(* Schneider Machine Expert - Basic project Slave 1 AHU Mod  TCP, file version 2.2.0.0 *)
(* ProjectInformations: Name=New project *)

HARDWARE
  Cpu 0: TM221ME16R/G
  ModuleExtensionObject 0: TM3DI16/G
  ModuleExtensionObject 1: TM3DQ16R/G
  ModuleExtensionObject 2: TM3AI8/G
  ModuleExtensionObject 3: TM3AQ4/G
  ModuleExtensionObject 4: TM3AQ2/G
  EthernetConfiguration: NetworkName=M221, IpAllocationMode=FixedAddress, IpAddress=10.3.12.251, SubnetMask=255.255.252.0
  SerialLineConfiguration: Baud=Baud9600, Parity=ParityEven, DataBits=DataBits8, StopBits=StopBits1, PhysicalMedium=PhysicalMediumRs485, TransmissionMode=TransmissionModeModbusRtu, SlaveId=1, Addressing=MasterAddressing
  MastTask: UsePeriodScanMode=false, PeriodScan=100
  FastTask: Period=255
  CpuBehavior: StartingMode=StartAsPreviousState, AutoSaveRamOnEeprom=true, WatchdogPeriod=250

SYMBOLS  (address, symbol, comment, settings)
  %M0       STRINV1  "Start Inverter AHU Line 09-10"
  %M1       STPINV1  "Stop Inverter AHU Line 09-10"
  %M2       OPNDMPR1  "Open Damper AHU Line 09-10"
  %M3       CLODMPR1  "Close Damper AHU Line 09-10"
  %M4       S_REMOTE_1  "Selector REMOTE MODE !!! Line 09-10"
  %M5       S_LOCAL_1  "Selector LOCAL MODE !!! Line 09-10"
  %M6       STRINV2  "Start Inverter AHU Line 11-12"
  %M7       STPINV2  "Stop Inverter AHU Line 11-12"
  %M8       OPNDMPR2  "Open Damper AHU Line 11-12"
  %M9       CLODMPR2  "Close Damper AHU Line 11-12"
  %M10      S_REMOTE_2  "Selector REMOTE MODE !!! Line 11-12"
  %M11      STRINV3  "Start Inverter AHU Line 17-18"
  %M12      STPINV3  "Stop Inverter AHU Line 17-18"
  %M13      OPNDMPR3  "Open Damper AHU Line 17-18"
  %M14      CLODMPR3  "Close Damper AHU Line 17-18"
  %M15      S_REMOTE_3  "Selector REMOTE MODE !!! Line 17-18"
  %M16      INPUT_ONINV_1  "On Inverter AHU Line 09-10"
  %M17      INPUT_ONINV_2  "On Inverter AHU Line 11-12"
  %M18      INPUT_ONINV_3  "On Inverter AHU Line 17-18"
  %M19      INPUT_ALARM_1  "Alarm Inverter AHU Line 09-10"
  %M20      INPUT_ALARM_2  "Alarm Inverter AHU Line 11-12"
  %M21      INPUT_ALARM_3  "Alarm Inverter AHU Line 17-18"
  %M22      S_LOCAL_2  "Selector LOCAL MODE !!! Line 11-12"
  %M23      S_LOCAL_3  "Selector LOCAL MODE !!! Line 17-18"
  %M31      ALARM1  "ALARM AHU LINE 09-10 ON !!!!"
  %M32      ALARM2  "ALARM AHU LINE 11-12 ON !!!!"
  %M33      ALARM3  "ALARM AHU LINE 17-18 ON !!!!"
  %M34      RUN_1  "RUN AHU LINE 09-10"
  %M35      RUN_2  "RUN AHU LINE 11-12"
  %M36      RUN_3  "RUN AHU LINE 17-18"
  %M37      INV_1_ON  "INVERTER AHU LINE 09-10 ON !!!"
  %M38      INV_2_ON  "INVERTER AHU LINE 11-12 ON !!!"
  %M39      INV_3_ON  "INVERTER AHU LINE 17-18 ON !!!"
  %M61      FLAG_MAN_INV1  "INVERTER LINE 09-10 ON !!! MANUAL"
  %M62      FLAG_MAN_DMPR1  "DAMPER LINE 09-10 ON !!! MANUAL"
  %M63      FLAG_AUTO_INV1  "INVERTER LINE 09-10 ON !!! AUTO"
  %M64      FLAG_MAN_INV2  "INVERTER LINE 11-12 ON !!! MANUAL"
  %M65      FLAG_MAN_DMPR2  "DAMPER LINE 11-12 ON !!! MANUAL"
  %M66      FLAG_AUTO_INV2  "INVERTER LINE 11-12 ON !!! AUTO"
  %M67      FLAG_MAN_INV3  "INVERTER LINE 17-18 ON !!! MANUAL"
  %M68      FLAG_MAN_DMPR3  "DAMPER LINE 17-18 ON !!! MANUAL"
  %M69      FLAG_AUTO_INV3  "INVERTER LINE 17-18 ON !!! AUTO"
  %M82      FLAG_AUTO_DMPR_1  "DAMPER LINE 09-10 ON !!! AUTO"
  %M83      FLAG_AUTO_DMPR_2  "DAMPER LINE 11-12 ON !!! AUTO"
  %M84      FLAG_AUTO_DMPR_3  "DAMPER LINE 17-18 ON !!! AUTO"
  %M85      ALARM_MODBUS  "MODBUS COMMUNICATION ERROR !!! CHECK CONNECTION"
  %M86      REMOTE_START_INV_1  "REMOTE Start Inverter AHU Line 09-10"
  %M87      REMOTE_STOP_INV_1  "REMOTE Stop Inverter AHU Line 09-10"
  %M88      REMOTE_START_DMPR_1  "REMOTE Open Damper AHU Line 09-10"
  %M89      REMOTE_STOP_DMPR_1  "REMOTE Close Damper AHU Line 09-10"
  %M90      REMOTE_START_INV_2  "REMOTE Start Inverter AHU Line 11-12"
  %M91      REMOTE_STOP_INV_2  "REMOTE Stop Inverter AHU Line 11-12"
  %M92      REMOTE_START_DMPR_2  "REMOTE Open Damper AHU Line 11-12"
  %M93      REMOTE_STOP_DMPR_2  "REMOTE Close Damper AHU Line 11-12"
  %M94      REMOTE_START_INV_3  "REMOTE Start Inverter AHU Line 17-18"
  %M95      REMOTE_STOP_INV_3  "REMOTE Stop Inverter AHU Line 17-18"
  %M96      REMOTE_START_DMPR_3  "REMOTE Open Damper AHU Line 17-18"
  %M97      REMOTE_STOP_DMPR_3  "REMOTE Close Damper AHU Line 17-18"
  %M100     MANUAL_AUTO_1  "REMOTE OPTION MODE AHU LINE 09-10"
  %M101     MANUAL_AUTO_2  "REMOTE OPTION MODE AHU LINE 11-12"
  %M102     MANUAL_AUTO_3  "REMOTE OPTION MODE AHU LINE 17-18"
  %M103     DMPR_1_ON  "DAMPER LINE 09-10 ON !!!"
  %M104     DMPR_2_ON  "DAMPER LINE 11-12 ON !!!"
  %M105     DMPR_3_ON  "DAMPER LINE 17-18 ON !!!"
  %M106     ERR_SERIAL_1  "Serial Comunication Error 1"
  %M107     ERR_SERIAL_2  "Serial Communication Error 2"
  %M119     RESET_ALARM
  %M120     TEMP_1_HIGH
  %M121     TEMP_1_LOW
  %M122     HUM_1_HIGH
  %M123     HUM_1_LOW
  %M124     PRESS_1_HIGH
  %M125     PRESS_1_LOW
  %M130     TEMP_2_HIGH
  %M131     TEMP_2_LOW
  %M132     HUM_2_HIGH
  %M133     HUM_2_LOW
  %M134     PRESS_2_HIGH
  %M135     PRESS_2_LOW
  %M140     TEMP_3_HIGH
  %M141     TEMP_3_LOW
  %M142     HUM_3_HIGH
  %M143     HUM_3_LOW
  %M144     PRESS_3_HIGH
  %M145     PRESS_3_LOW
  %S6       SB_TB1S  "Time base of 1 s generated by an internal clock"
  %S12      SB_RUNMODE  "The controller is running"
  %MW9      AI_SCALE_DIFF_PRESSURE_1  "Memory Hasil Scalling Analog Input Differensial Pressure Line 09-10"
  %MW11     AO1_LO_LIMIT
  %MW12     AO1_HI_LIMIT
  %MW13     AO2_LO_LIMIT
  %MW14     AO2_HI_LIMIT
  %MW15     AO3_LO_LIMIT
  %MW16     AO3_HI_LIMIT
  %MW30     AI_SCALE_DIFF_PRESSURE_2
  %MW51     AI_SCALE_DIFF_PRESSURE_3
  %MW73     AI_SCALE_TEMP_1
  %MW95     AI_SCALE_HUMIDITY_1
  %MW117    AO_SCALE_TEMP_1
  %MW139    AO_SCALE_TEMP_2
  %MW161    AO_SCALE_TEMP_3
  %MW183    AO_SCALE_HUMIDITY_1
  %MW205    AO_SCALE_HUMIDITY_2
  %MW227    AO_SCALE_HUMIDITY_3
  %MW251    TEMP_1_SETPOINT
  %MW252    TEMP_1_P
  %MW253    TEMP_1_I
  %MW254    TEMP_1_D
  %MW255    TEMP_1_SAMPLING
  %MW256    SET_SPEED_INV_1
  %MW257    ALRM_TEMP1_LOW_SET
  %MW258    ALRM_TEMP1_HIGH_SET
  %MW259    ALRM_PRESS1_LOW_SET
  %MW260    ALRM_PRESS1_HIGH_SET
  %MW281    TEMP_2_SETPOINT
  %MW282    TEMP_2_P
  %MW283    TEMP_2_I
  %MW284    TEMP_2_D
  %MW285    TEMP_2_SAMPLING
  %MW286    SET_SPEED_INV_2
  %MW287    ALRM_TEMP_2_LOW_SET
  %MW288    ALRM_TEMP_2_HIGH_SET
  %MW289    ALRM_PRESS2_LOW_SET
  %MW290    ALRM_PRESS2_HIGH_SET
  %MW311    TEMP_3_SETPOINT
  %MW312    TEMP_3_P
  %MW313    TEMP_3_I
  %MW314    TEMP_3_D
  %MW315    TEMP_3_SAMPLING
  %MW316    SET_SPEED_INV_3
  %MW317    ALRM_TEMP_3_LOW_SET
  %MW318    ALRM_TEMP_3_HIGH_SET
  %MW319    ALRM_PRESS3_LOW_SET
  %MW320    ALRM_PRESS3_HIGH_SET
  %MW341    HUMIDITY_1_SETPOINT
  %MW342    HUMIDITY_1_P
  %MW343    HUMIDITY_1_I
  %MW344    HUMIDITY_1_D
  %MW345    HUMIDITY_1_SAMPLING
  %MW346    SET_DAMPER_POSITION_1
  %MW347    ALRM_HUMIDITY_1_LOW_SET
  %MW348    ALRM_HUMIDITY_1_HIGH_SET
  %MW380    DMPR_1_VIEW
  %MW381    DMPR_2_VIEW
  %MW382    DMPR_3_VIEW
  %MW401    HUMIDITY_2_SETPOINT
  %MW402    HUMIDITY_2_P
  %MW403    HUMIDITY_2_I
  %MW404    HUMIDITY_2_D
  %MW405    HUMIDITY_2_SAMPLING
  %MW406    SET_DAMPER_2_POSITION
  %MW407    ALRM_HUMIDITY_2_LOW_SET
  %MW408    ALRM_HUMIDITY_2_HIGH_SET
  %MW431    HUMIDITY_3_SETPOINT
  %MW432    HUMIDITY_3_P
  %MW433    HUMIDITY_3_I
  %MW434    HUMIDITY_3_D
  %MW435    HUMIDITY_3_SAMPLING
  %MW436    SET_DAMPER_3_POSITION
  %MW437    ALRM_HUMIDITY_3_LOW_SET
  %MW438    ALRM_HUMIDITY_3_HIGH_SET
  %MW461    TEMP_1_DATA_SERIAL  "Data Temperature Line 09-10"
  %MW462    TEMP_2_DATA_SERIAL  "Data Temperature Line 11-12"
  %MW463    HUMIDITY_1_DATA_SERIAL  "Data Humidity Line 09-10"
  %MW464    HUMIDITY_2_DATA_SERIAL  "Data Humidity Line 11-12"
  %MW465    ERROR_DATA  "Error Communication"
  %MW480    AI_SCALE_TEMP_2
  %MW490    AI_SCALE_TEMP_3
  %MW500    AI_SCALE_HUMIDITY_2
  %MW510    AI_SCALE_HUMIDITY_3
  %MW520    AI_SCALE_DAMPER__POSITION_1
  %MW530    AI_SCALE_DAMPER_POSITION_2
  %MW540    AI_SCALE_DAMPER_POSITION_3
  %MW542    ALARM_WORD
  %MW600    HUMIDITY_LINE_1718  "Data serial humidity line 17-18"
  %MW601    TEMPERATURE_LINE_1718  "Data serial temperature line 17-18"
  %MW630    INV_1_HZ
  %MW640    INV_2_HZ
  %MW650    INV_3_HZ
  %READ_VAR0   [Link(Value(FBComLinkParameterEnums=SerialLine1)), RemoteDeviceId(Value(int=2)), Timeout(Value(int=100)), ObjType(Value(FBComObjTypeParameterEnums=IW)), FirstObj(Value(int=0)), Quantity(Value(int=1)), IndexData(Value(int=600))]
  %READ_VAR1   [Link(Value(FBComLinkParameterEnums=SerialLine1)), RemoteDeviceId(Value(int=3)), Timeout(Value(int=100)), ObjType(Value(FBComObjTypeParameterEnums=IW)), FirstObj(Value(int=0)), Quantity(Value(int=1)), IndexData(Value(int=601))]
  %RTC0     REAL_TIME_0  [Day(Value(int=1)), Month(Value(int=1)), Year(Value(int=2000)), Hours(Value(int=0)), Minutes(Value(int=0)), Seconds(Value(int=0))]
  %WRITE_READ_VAR0   [Link(Value(FBComLinkParameterEnums=EthernetLink)), RemoteDeviceId(Value(int=1)), Timeout(Value(int=100)), ObjType(Value(FBComObjTypeParameterEnums=MW)), FirstWriteObj(Value(int=10)), WriteQuantity(Value(int=1)), IndexDataOut(Value(int=465)), FirstReadObj(Value(int=0)), ReadQuantity(Value(int=4)), IndexDataIn(Value(int=461))]
  %I0.0     INV1_START  "LOCAL !!! Untuk mengontrol START Inverter AHU Line 09-10"
  %I0.1     INV1_STOP  "LOCAL !!! Untuk mengontrol STOP Inverter AHU Line 09-10"
  %I0.2     DMPR1_OPEN  "LOCAL !!! Untuk mengontrol OPEN Damper  AHU Line 09-10"
  %I0.3     DMPR1_CLOSE  "LOCAL !!! Untuk mengontrol CLOSE Damper  AHU Line 09-10"
  %I0.4     REMOTE_1  "SELECTOR SWITCH REMOTE !!! AHU LINE 09-10"
  %I0.5     LOCAL_1  "SELECTOR SWITCH LOCAL !!! AHU LINE 09-10"
  %I0.6     INV2_START  "LOCAL !!! Untuk mengontrol START Inverter AHU Line 11-12"
  %I0.7     INV2_STOP  "LOCAL !!! Untuk mengontrol STOP Inverter AHU Line 11-12"
  %Q0.0     ALARM_1  "Alarm Indikator Line 09-10"
  %Q0.1     ALARM_2  "Alarm Indikator Line 11-12"
  %Q0.2     ALARM_3  "Alarm Indikator Line 17-18"
  %Q0.3     RUN_STATUS_1  "Running Status Line 09-10"
  %Q0.4     RUN_STATUS_2  "Running Status Line 11-12"
  %Q0.5     RUN_STATUS_3  "Running Status Line 17-18"
  %Q0.6     INVERTER_1_ON  "Trigger Inverter Line 09-10"
  %Q0.7     INVERTER_2_ON  "Trigger Inverter Line 11-12"
  %I1.0     DMPR2_OPEN  "LOCAL !!! Untuk mengontrol OPEN Damper  AHU Line 11-12"
  %I1.1     DMPR2_CLOSE  "LOCAL !!! Untuk mengontrol CLOSE Damper  AHU Line 11-12"
  %I1.2     REMOTE_2  "SELECTOR SWITCH REMOTE !!! AHU LINE 11-12"
  %I1.3     INV3_START  "LOCAL !!! Untuk mengontrol START Inverter AHU Line 17-18"
  %I1.4     INV3_STOP  "LOCAL !!! Untuk mengontrol STOP Inverter AHU Line  17-18"
  %I1.5     DMPR3_OPEN  "LOCAL !!! Untuk mengontrol OPEN Damper  AHU Line 17-18"
  %I1.6     DMPR3_CLOSE  "LOCAL !!! Untuk mengontrol CLOSE Damper  AHU Line 17-18"
  %I1.7     REMOTE_3  "SELECTOR SWITCH REMOTE !!! AHU LINE 17-18"
  %I1.8     INPUTRUN1  "Signal Running Inverter AHU Line 09-10"
  %I1.9     INPUTRUN2  "Signal Running Inverter AHU Line 11-12"
  %I1.10    INPUTRUN3  "Signal Running Inverter AHU Line 17-18"
  %I1.11    ALARM1_INPUT  "Signal Alarm Inverter AHU Line 09-10"
  %I1.12    ALARM2_INPUT  "Signal Alarm Inverter AHU Line 11-12"
  %I1.13    ALARM3_INPUT  "Signal Alarm Inverter AHU Line 17-18"
  %I1.14    LOCAL_2  "SELECTOR SWITCH LOCAL !!! AHU LINE 11-12"
  %I1.15    LOCAL_3  "SELECTOR SWITCH LOCAL !!! AHU LINE 17-18"
  %Q2.0     INVERTER_3_ON  "Trigger Inverter Line 17-18"
  %IW3.0    PRESS_AHU_1  "Differensial Pressure Line 09-10"  [Type=Type_4_20mA, Scope=Scope_Customized, Minimum=4000, Maximum=20000]
  %IW3.1    PRESS_AHU_2  "Differensial Pressure Line 11-12"  [Type=Type_4_20mA, Scope=Scope_Customized, Minimum=4000, Maximum=20000]
  %IW3.2    PRESS_AHU_3  "Differensial Pressure Line 17-18"  [Type=Type_4_20mA, Scope=Scope_Customized, Minimum=4000, Maximum=20000]
  %IW3.3    SPARE1  [Type=Type_4_20mA, Scope=Scope_Customized, Minimum=4000, Maximum=20000]
  %IW3.4    SPARE2  [Type=Type_4_20mA, Scope=Scope_Customized, Minimum=4000, Maximum=20000]
  %IW3.5    DAMP_POS_AHU_1  "FeedBack Damper Position Line 09-10"  [Type=Type_0_10V, Scope=Scope_Customized, Minimum=0, Maximum=10000]
  %IW3.6    DAMP_POS_AHU_2  "FeedBack Damper Position Line 11-12"  [Type=Type_0_10V, Scope=Scope_Customized, Minimum=0, Maximum=10000]
  %IW3.7    DAMP_POS_AHU_3  "FeedBack Damper Position Line 17-18"  [Type=Type_0_10V, Scope=Scope_Customized, Minimum=0, Maximum=10000]
  %QW4.0    AO_INV_1  "Analog Output Speed Inverter Line 09-10"  [Type=Type_0_10V, Scope=Scope_Customized, Minimum=0, Maximum=10000]
  %QW4.1    AO_INV_2  "Analog Output Speed Inverter Line 11-12"  [Type=Type_0_10V, Scope=Scope_Customized, Minimum=0, Maximum=10000]
  %QW4.2    AO_INV_3  "Analog Output Speed Inverter Line 17-18"  [Type=Type_0_10V, Scope=Scope_Customized, Minimum=0, Maximum=10000]
  %QW4.3    AO_DMPR_1  "Analog Output Damper Control Line 09-10"  [Type=Type_0_10V, Scope=Scope_Customized, Minimum=0, Maximum=10000]
  %QW5.0    AO_DMPR_2  "Analog Output Damper Control Line 11-12"  [Type=Type_0_10V, Scope=Scope_Customized, Minimum=0, Maximum=10000]
  %QW5.1    AO_DMPR_3  "Analog Output Damper Control Line 17-18"  [Type=Type_0_10V, Scope=Scope_Customized, Minimum=0, Maximum=10000]

POU TRANSFER INPUT OUTPUT
  (* SectionNumber=1 *)

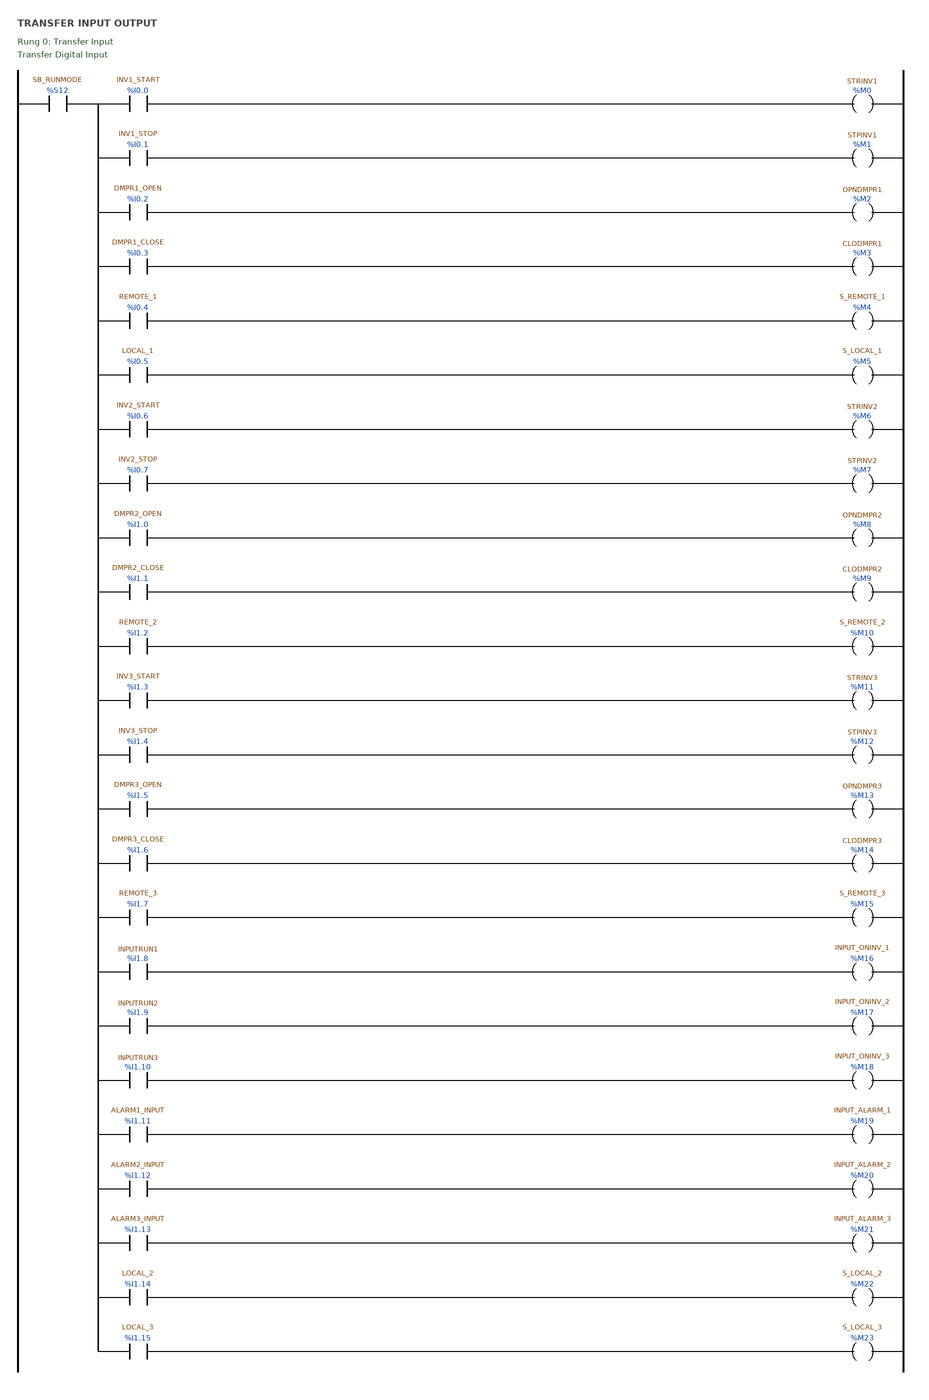

// Rung 0: Transfer Input
// Transfer Digital Input
  LD %S12                 (* SB_RUNMODE *)
  MPS
  AND %I0.0               (* INV1_START *)
  ST %M0                  (* STRINV1 *)
  MRD
  AND %I0.1               (* INV1_STOP *)
  ST %M1                  (* STPINV1 *)
  MRD
  AND %I0.2               (* DMPR1_OPEN *)
  ST %M2                  (* OPNDMPR1 *)
  MRD
  AND %I0.3               (* DMPR1_CLOSE *)
  ST %M3                  (* CLODMPR1 *)
  MRD
  AND %I0.4               (* REMOTE_1 *)
  ST %M4                  (* S_REMOTE_1 *)
  MRD
  AND %I0.5               (* LOCAL_1 *)
  ST %M5                  (* S_LOCAL_1 *)
  MRD
  AND %I0.6               (* INV2_START *)
  ST %M6                  (* STRINV2 *)
  MRD
  AND %I0.7               (* INV2_STOP *)
  ST %M7                  (* STPINV2 *)
  MRD
  AND %I1.0               (* DMPR2_OPEN *)
  ST %M8                  (* OPNDMPR2 *)
  MRD
  AND %I1.1               (* DMPR2_CLOSE *)
  ST %M9                  (* CLODMPR2 *)
  MRD
  AND %I1.2               (* REMOTE_2 *)
  ST %M10                 (* S_REMOTE_2 *)
  MRD
  AND %I1.3               (* INV3_START *)
  ST %M11                 (* STRINV3 *)
  MRD
  AND %I1.4               (* INV3_STOP *)
  ST %M12                 (* STPINV3 *)
  MRD
  AND %I1.5               (* DMPR3_OPEN *)
  ST %M13                 (* OPNDMPR3 *)
  MRD
  AND %I1.6               (* DMPR3_CLOSE *)
  ST %M14                 (* CLODMPR3 *)
  MRD
  AND %I1.7               (* REMOTE_3 *)
  ST %M15                 (* S_REMOTE_3 *)
  MRD
  AND %I1.8               (* INPUTRUN1 *)
  ST %M16                 (* INPUT_ONINV_1 *)
  MRD
  AND %I1.9               (* INPUTRUN2 *)
  ST %M17                 (* INPUT_ONINV_2 *)
  MRD
  AND %I1.10              (* INPUTRUN3 *)
  ST %M18                 (* INPUT_ONINV_3 *)
  MRD
  AND %I1.11              (* ALARM1_INPUT *)
  ST %M19                 (* INPUT_ALARM_1 *)
  MRD
  AND %I1.12              (* ALARM2_INPUT *)
  ST %M20                 (* INPUT_ALARM_2 *)
  MRD
  AND %I1.13              (* ALARM3_INPUT *)
  ST %M21                 (* INPUT_ALARM_3 *)
  MRD
  AND %I1.14              (* LOCAL_2 *)
  ST %M22                 (* S_LOCAL_2 *)
  MPP
  AND %I1.15              (* LOCAL_3 *)
  ST %M23                 (* S_LOCAL_3 *)
  // as ST:
  //   STRINV1 := SB_RUNMODE AND INV1_START;
  //   STPINV1 := SB_RUNMODE AND INV1_STOP;
  //   OPNDMPR1 := SB_RUNMODE AND DMPR1_OPEN;
  //   CLODMPR1 := SB_RUNMODE AND DMPR1_CLOSE;
  //   S_REMOTE_1 := SB_RUNMODE AND REMOTE_1;
  //   S_LOCAL_1 := SB_RUNMODE AND LOCAL_1;
  //   STRINV2 := SB_RUNMODE AND INV2_START;
  //   STPINV2 := SB_RUNMODE AND INV2_STOP;
  //   OPNDMPR2 := SB_RUNMODE AND DMPR2_OPEN;
  //   CLODMPR2 := SB_RUNMODE AND DMPR2_CLOSE;
  //   S_REMOTE_2 := SB_RUNMODE AND REMOTE_2;
  //   STRINV3 := SB_RUNMODE AND INV3_START;
  //   STPINV3 := SB_RUNMODE AND INV3_STOP;
  //   OPNDMPR3 := SB_RUNMODE AND DMPR3_OPEN;
  //   CLODMPR3 := SB_RUNMODE AND DMPR3_CLOSE;
  //   S_REMOTE_3 := SB_RUNMODE AND REMOTE_3;
  //   INPUT_ONINV_1 := SB_RUNMODE AND INPUTRUN1;
  //   INPUT_ONINV_2 := SB_RUNMODE AND INPUTRUN2;
  //   INPUT_ONINV_3 := SB_RUNMODE AND INPUTRUN3;
  //   INPUT_ALARM_1 := SB_RUNMODE AND ALARM1_INPUT;
  //   INPUT_ALARM_2 := SB_RUNMODE AND ALARM2_INPUT;
  //   INPUT_ALARM_3 := SB_RUNMODE AND ALARM3_INPUT;
  //   S_LOCAL_2 := SB_RUNMODE AND LOCAL_2;
  //   S_LOCAL_3 := SB_RUNMODE AND LOCAL_3;

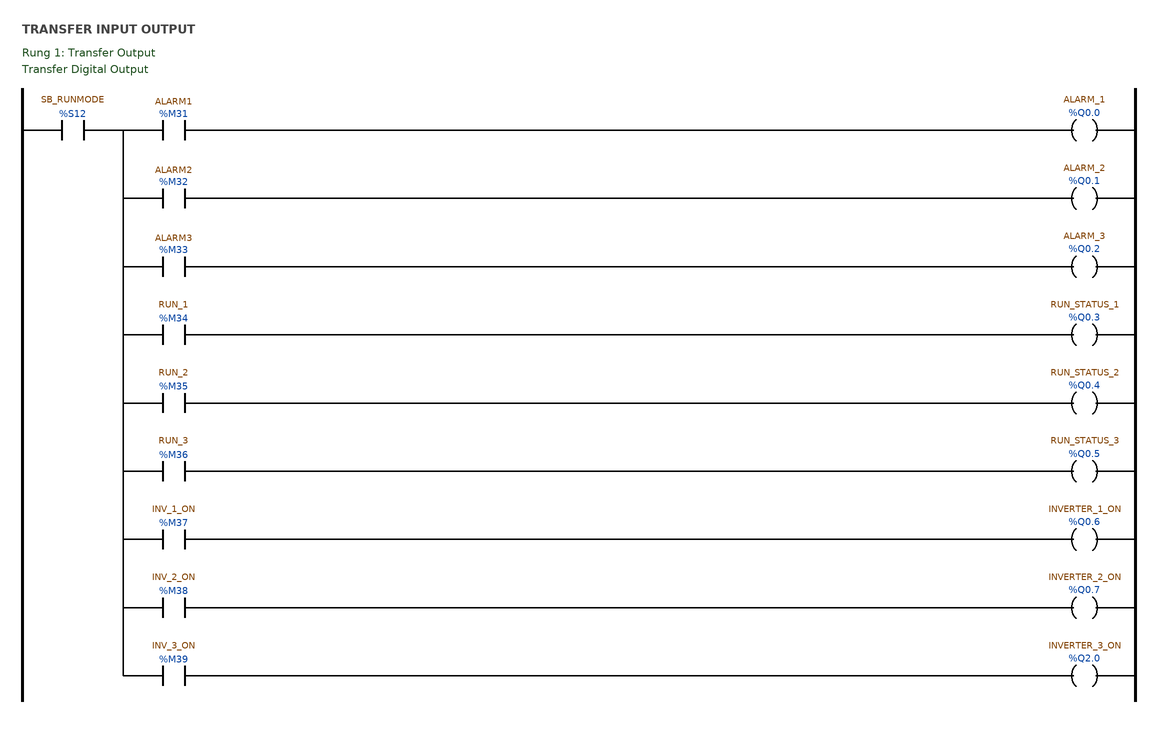

// Rung 1: Transfer Output
// Transfer Digital Output
  LD %S12                 (* SB_RUNMODE *)
  MPS
  AND %M31                (* ALARM1 *)
  ST %Q0.0                (* ALARM_1 *)
  MRD
  AND %M32                (* ALARM2 *)
  ST %Q0.1                (* ALARM_2 *)
  MRD
  AND %M33                (* ALARM3 *)
  ST %Q0.2                (* ALARM_3 *)
  MRD
  AND %M34                (* RUN_1 *)
  ST %Q0.3                (* RUN_STATUS_1 *)
  MRD
  AND %M35                (* RUN_2 *)
  ST %Q0.4                (* RUN_STATUS_2 *)
  MRD
  AND %M36                (* RUN_3 *)
  ST %Q0.5                (* RUN_STATUS_3 *)
  MRD
  AND %M37                (* INV_1_ON *)
  ST %Q0.6                (* INVERTER_1_ON *)
  MRD
  AND %M38                (* INV_2_ON *)
  ST %Q0.7                (* INVERTER_2_ON *)
  MPP
  AND %M39                (* INV_3_ON *)
  ST %Q2.0                (* INVERTER_3_ON *)
  // as ST:
  //   ALARM_1 := SB_RUNMODE AND ALARM1;
  //   ALARM_2 := SB_RUNMODE AND ALARM2;
  //   ALARM_3 := SB_RUNMODE AND ALARM3;
  //   RUN_STATUS_1 := SB_RUNMODE AND RUN_1;
  //   RUN_STATUS_2 := SB_RUNMODE AND RUN_2;
  //   RUN_STATUS_3 := SB_RUNMODE AND RUN_3;
  //   INVERTER_1_ON := SB_RUNMODE AND INV_1_ON;
  //   INVERTER_2_ON := SB_RUNMODE AND INV_2_ON;
  //   INVERTER_3_ON := SB_RUNMODE AND INV_3_ON;

POU AHU LINE 09-10
  (* SectionNumber=2 *)

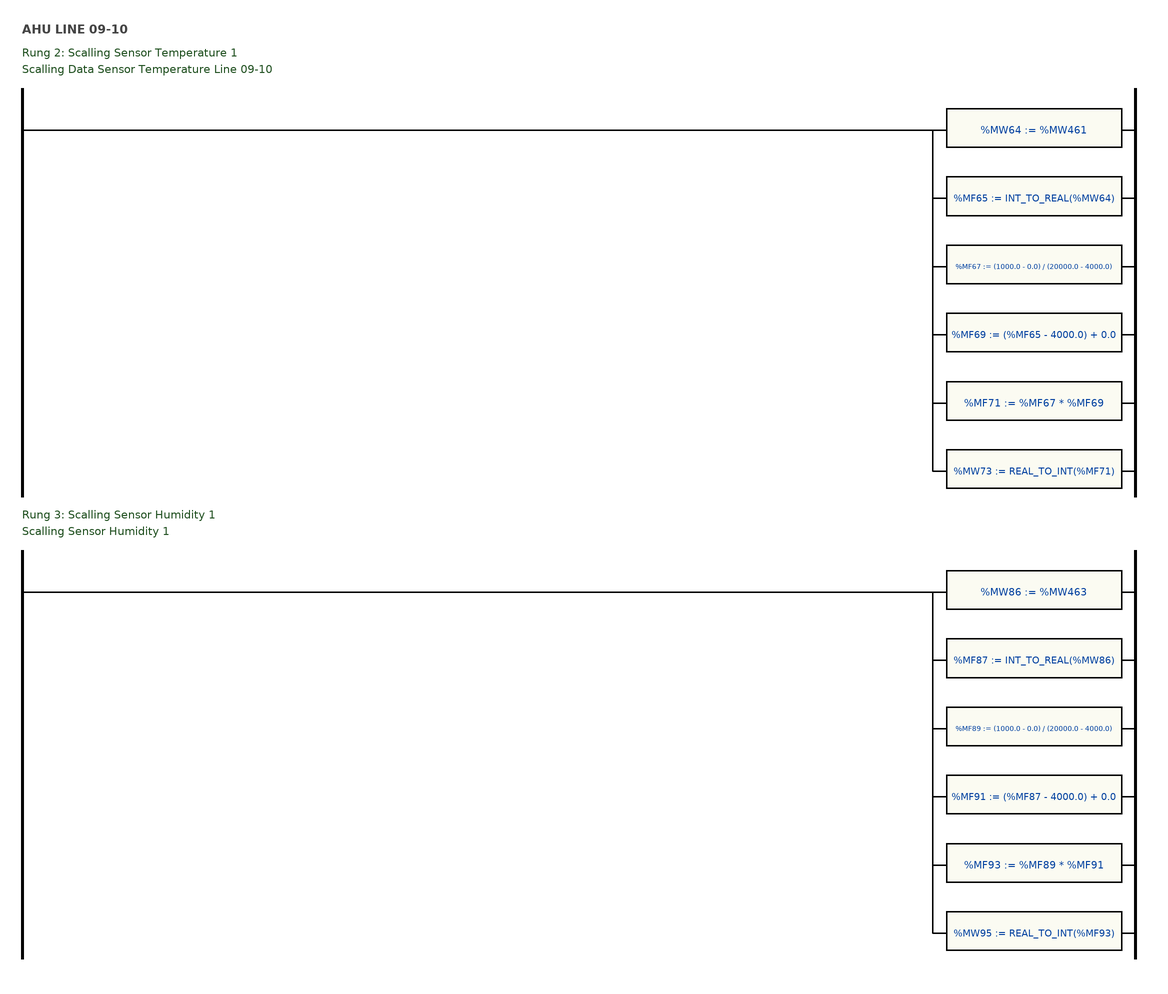

// Rung 2: Scalling Sensor Temperature 1
// Scalling Data Sensor Temperature Line 09-10
  LD 1
  [ %MW64 := %MW461 ]     (* TEMP_1_DATA_SERIAL *)
  [ %MF65 := INT_TO_REAL ( %MW64 ) ]
  [%MF67 := (1000.0 - 0.0) / (20000.0 - 4000.0)]
  [%MF69 := (%MF65 - 4000.0) + 0.0]
  [ %MF71 := %MF67 * %MF69 ]
  [ %MW73 := REAL_TO_INT ( %MF71 ) ](* AI_SCALE_TEMP_1 *)
  // as ST:
  //   %MW64 := TEMP_1_DATA_SERIAL;
  //   %MF65 := INT_TO_REAL ( %MW64 );
  //   %MF67 := (1000.0 - 0.0) / (20000.0 - 4000.0);
  //   %MF69 := (%MF65 - 4000.0) + 0.0;
  //   %MF71 := %MF67 * %MF69;
  //   AI_SCALE_TEMP_1 := REAL_TO_INT ( %MF71 );

// Rung 3: Scalling Sensor Humidity 1
// Scalling Sensor Humidity 1
  LD 1
  [ %MW86 := %MW463 ]     (* HUMIDITY_1_DATA_SERIAL *)
  [ %MF87 := INT_TO_REAL ( %MW86 ) ]
  [%MF89 := (1000.0 - 0.0) / (20000.0 - 4000.0)]
  [%MF91 := (%MF87 - 4000.0) + 0.0]
  [ %MF93 := %MF89 * %MF91 ]
  [ %MW95 := REAL_TO_INT ( %MF93 ) ](* AI_SCALE_HUMIDITY_1 *)
  // as ST:
  //   %MW86 := HUMIDITY_1_DATA_SERIAL;
  //   %MF87 := INT_TO_REAL ( %MW86 );
  //   %MF89 := (1000.0 - 0.0) / (20000.0 - 4000.0);
  //   %MF91 := (%MF87 - 4000.0) + 0.0;
  //   %MF93 := %MF89 * %MF91;
  //   AI_SCALE_HUMIDITY_1 := REAL_TO_INT ( %MF93 );

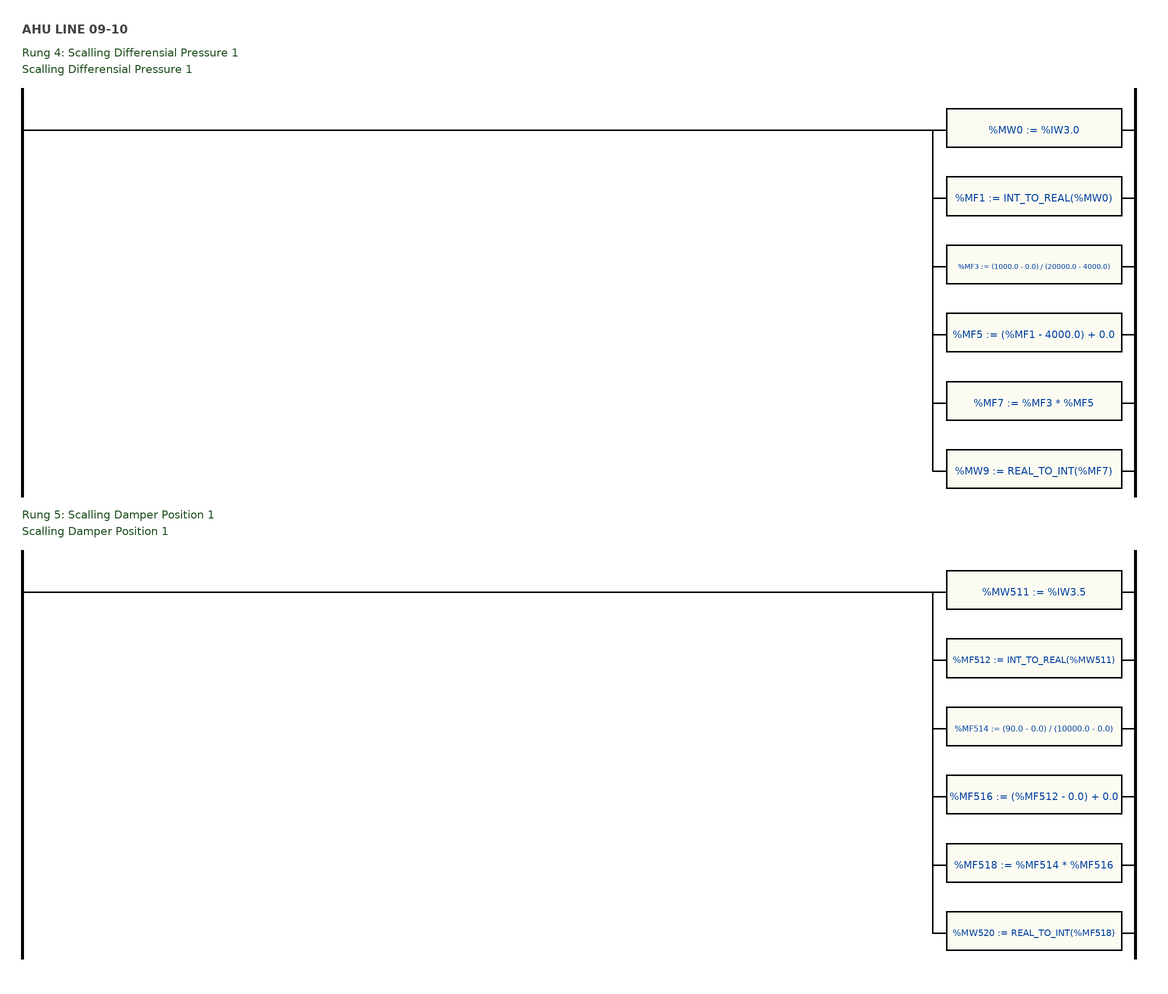

// Rung 4: Scalling Differensial Pressure 1
// Scalling Differensial Pressure 1
  LD 1
  [ %MW0 := %IW3.0 ]      (* PRESS_AHU_1 *)
  [ %MF1 := INT_TO_REAL ( %MW0 ) ]
  [%MF3 := (1000.0 - 0.0) / (20000.0 - 4000.0)]
  [%MF5 := (%MF1 - 4000.0) + 0.0]
  [ %MF7 := %MF3 * %MF5 ]
  [ %MW9 := REAL_TO_INT ( %MF7 ) ](* AI_SCALE_DIFF_PRESSURE_1 *)
  // as ST:
  //   %MW0 := PRESS_AHU_1;
  //   %MF1 := INT_TO_REAL ( %MW0 );
  //   %MF3 := (1000.0 - 0.0) / (20000.0 - 4000.0);
  //   %MF5 := (%MF1 - 4000.0) + 0.0;
  //   %MF7 := %MF3 * %MF5;
  //   AI_SCALE_DIFF_PRESSURE_1 := REAL_TO_INT ( %MF7 );

// Rung 5: Scalling Damper Position 1
// Scalling Damper Position 1
  LD 1
  [ %MW511 := %IW3.5 ]    (* DAMP_POS_AHU_1 *)
  [ %MF512 := INT_TO_REAL ( %MW511 ) ]
  [%MF514 := (90.0 - 0.0) / (10000.0 - 0.0)]
  [%MF516 := (%MF512 - 0.0) + 0.0]
  [ %MF518 := %MF514 * %MF516 ]
  [ %MW520 := REAL_TO_INT ( %MF518 ) ](* AI_SCALE_DAMPER__POSITION_1 *)
  // as ST:
  //   %MW511 := DAMP_POS_AHU_1;
  //   %MF512 := INT_TO_REAL ( %MW511 );
  //   %MF514 := (90.0 - 0.0) / (10000.0 - 0.0);
  //   %MF516 := (%MF512 - 0.0) + 0.0;
  //   %MF518 := %MF514 * %MF516;
  //   AI_SCALE_DAMPER__POSITION_1 := REAL_TO_INT ( %MF518 );

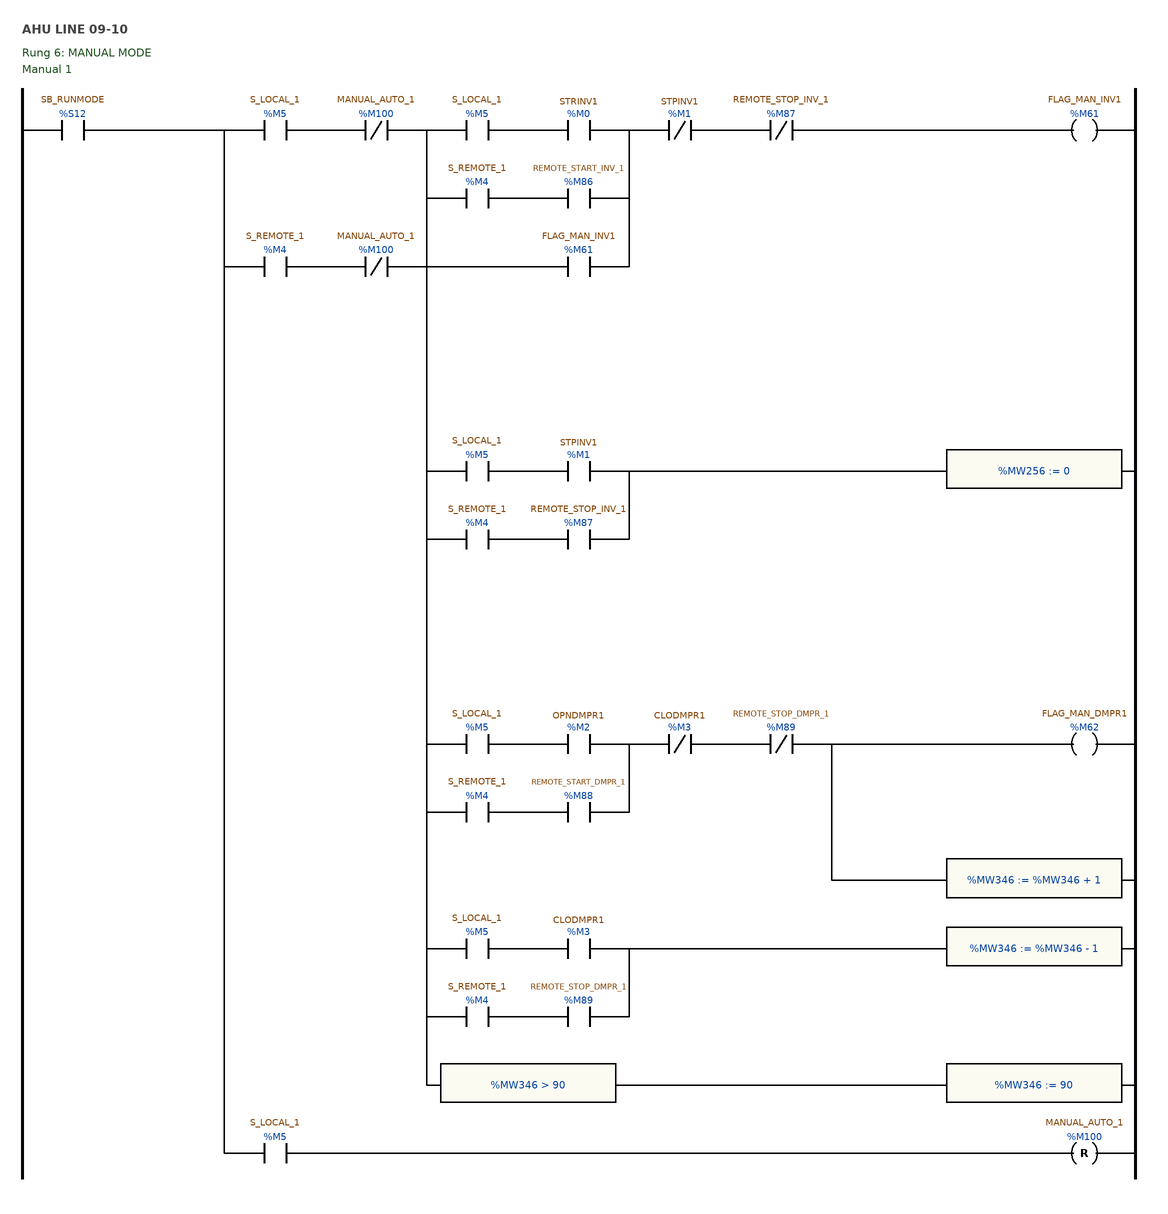

// Rung 6: MANUAL MODE
// Manual 1
  LD %S12                 (* SB_RUNMODE *)
  MPS
  AND( %M5                (* S_LOCAL_1 *)
  ANDN %M100              (* MANUAL_AUTO_1 *)
  OR( %M4                 (* S_REMOTE_1 *)
  ANDN %M100              (* MANUAL_AUTO_1 *)
  )
  )
  MPS
  AND( %M5                (* S_LOCAL_1 *)
  AND %M0                 (* STRINV1 *)
  OR( %M4                 (* S_REMOTE_1 *)
  AND %M86                (* REMOTE_START_INV_1 *)
  )
  OR %M61                 (* FLAG_MAN_INV1 *)
  )
  ANDN %M1                (* STPINV1 *)
  ANDN %M87               (* REMOTE_STOP_INV_1 *)
  ST %M61                 (* FLAG_MAN_INV1 *)
  MRD
  AND( %M5                (* S_LOCAL_1 *)
  AND %M1                 (* STPINV1 *)
  OR( %M4                 (* S_REMOTE_1 *)
  AND %M87                (* REMOTE_STOP_INV_1 *)
  )
  )
  [ %MW256 := 0 ]         (* SET_SPEED_INV_1 *)
  MRD
  AND( %M5                (* S_LOCAL_1 *)
  AND %M2                 (* OPNDMPR1 *)
  OR( %M4                 (* S_REMOTE_1 *)
  AND %M88                (* REMOTE_START_DMPR_1 *)
  )
  )
  ANDN %M3                (* CLODMPR1 *)
  ANDN %M89               (* REMOTE_STOP_DMPR_1 *)
  ST %M62                 (* FLAG_MAN_DMPR1 *)
  [ %MW346 := %MW346 + 1 ](* SET_DAMPER_POSITION_1, SET_DAMPER_POSITION_1 *)
  MRD
  AND( %M5                (* S_LOCAL_1 *)
  AND %M3                 (* CLODMPR1 *)
  OR( %M4                 (* S_REMOTE_1 *)
  AND %M89                (* REMOTE_STOP_DMPR_1 *)
  )
  )
  [ %MW346 := %MW346 - 1 ](* SET_DAMPER_POSITION_1, SET_DAMPER_POSITION_1 *)
  MPP
  AND [ %MW346 > 90 ]     (* SET_DAMPER_POSITION_1 *)
  [ %MW346 := 90 ]        (* SET_DAMPER_POSITION_1 *)
  MPP
  AND %M5                 (* S_LOCAL_1 *)
  R %M100                 (* MANUAL_AUTO_1 *)
  // as ST:
  //   FLAG_MAN_INV1 := SB_RUNMODE AND (S_LOCAL_1 AND NOT MANUAL_AUTO_1 OR S_REMOTE_1 AND NOT MANUAL_AUTO_1) AND (S_LOCAL_1 AND STRINV1 OR S_REMOTE_1 AND REMOTE_START_INV_1 OR FLAG_MAN_INV1) AND NOT STPINV1 AND NOT REMOTE_STOP_INV_1;
  //   IF SB_RUNMODE AND (S_LOCAL_1 AND NOT MANUAL_AUTO_1 OR S_REMOTE_1 AND NOT MANUAL_AUTO_1) AND (S_LOCAL_1 AND STPINV1 OR S_REMOTE_1 AND REMOTE_STOP_INV_1) THEN SET_SPEED_INV_1 := 0; END_IF;
  //   FLAG_MAN_DMPR1 := SB_RUNMODE AND (S_LOCAL_1 AND NOT MANUAL_AUTO_1 OR S_REMOTE_1 AND NOT MANUAL_AUTO_1) AND (S_LOCAL_1 AND OPNDMPR1 OR S_REMOTE_1 AND REMOTE_START_DMPR_1) AND NOT CLODMPR1 AND NOT REMOTE_STOP_DMPR_1;
  //   IF SB_RUNMODE AND (S_LOCAL_1 AND NOT MANUAL_AUTO_1 OR S_REMOTE_1 AND NOT MANUAL_AUTO_1) AND (S_LOCAL_1 AND OPNDMPR1 OR S_REMOTE_1 AND REMOTE_START_DMPR_1) AND NOT CLODMPR1 AND NOT REMOTE_STOP_DMPR_1 THEN SET_DAMPER_POSITION_1 := SET_DAMPER_POSITION_1 + 1; END_IF;
  //   IF SB_RUNMODE AND (S_LOCAL_1 AND NOT MANUAL_AUTO_1 OR S_REMOTE_1 AND NOT MANUAL_AUTO_1) AND (S_LOCAL_1 AND CLODMPR1 OR S_REMOTE_1 AND REMOTE_STOP_DMPR_1) THEN SET_DAMPER_POSITION_1 := SET_DAMPER_POSITION_1 - 1; END_IF;
  //   IF SB_RUNMODE AND (S_LOCAL_1 AND NOT MANUAL_AUTO_1 OR S_REMOTE_1 AND NOT MANUAL_AUTO_1) AND SET_DAMPER_POSITION_1 > 90 THEN SET_DAMPER_POSITION_1 := 90; END_IF;
  //   IF SB_RUNMODE AND S_LOCAL_1 THEN MANUAL_AUTO_1 := FALSE; END_IF;

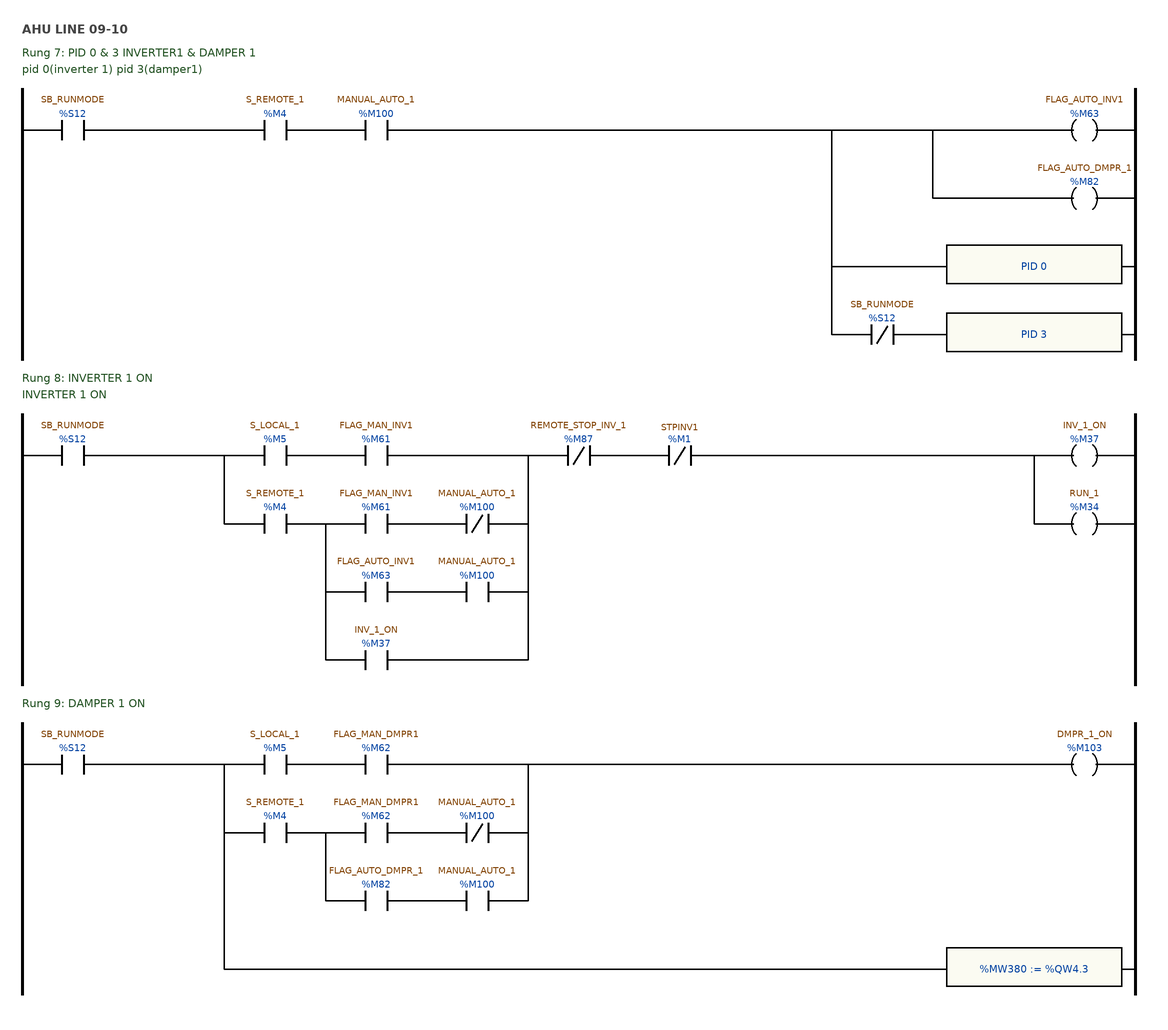

// Rung 7: PID 0 & 3 INVERTER1 & DAMPER 1
// pid 0(inverter 1) pid 3(damper1)
  LD %S12                 (* SB_RUNMODE *)
  AND %M4                 (* S_REMOTE_1 *)
  AND %M100               (* MANUAL_AUTO_1 *)
  MPS
  ST %M63                 (* FLAG_AUTO_INV1 *)
  ST %M82                 (* FLAG_AUTO_DMPR_1 *)
  MRD
  [ PID 0 ]
  MPP
  ANDN %S12               (* SB_RUNMODE *)
  [ PID 3 ]
  // as ST:
  //   FLAG_AUTO_INV1 := SB_RUNMODE AND S_REMOTE_1 AND MANUAL_AUTO_1;
  //   FLAG_AUTO_DMPR_1 := SB_RUNMODE AND S_REMOTE_1 AND MANUAL_AUTO_1;
  //   IF SB_RUNMODE AND S_REMOTE_1 AND MANUAL_AUTO_1 THEN PID 0; END_IF;
  //   IF SB_RUNMODE AND S_REMOTE_1 AND MANUAL_AUTO_1 AND NOT SB_RUNMODE THEN PID 3; END_IF;

// Rung 8: INVERTER 1 ON
// INVERTER 1 ON
  LD %S12                 (* SB_RUNMODE *)
  AND( %M5                (* S_LOCAL_1 *)
  AND %M61                (* FLAG_MAN_INV1 *)
  OR( %M4                 (* S_REMOTE_1 *)
  AND( %M61               (* FLAG_MAN_INV1 *)
  ANDN %M100              (* MANUAL_AUTO_1 *)
  OR( %M63                (* FLAG_AUTO_INV1 *)
  AND %M100               (* MANUAL_AUTO_1 *)
  )
  OR %M37                 (* INV_1_ON *)
  )
  )
  )
  ANDN %M87               (* REMOTE_STOP_INV_1 *)
  ANDN %M1                (* STPINV1 *)
  ST %M37                 (* INV_1_ON *)
  ST %M34                 (* RUN_1 *)
  // as ST:
  //   _t1 := SB_RUNMODE AND (S_LOCAL_1 AND FLAG_MAN_INV1 OR S_REMOTE_1 AND (FLAG_MAN_INV1 AND NOT MANUAL_AUTO_1 OR FLAG_AUTO_INV1 AND MANUAL_AUTO_1 OR INV_1_ON)) AND NOT REMOTE_STOP_INV_1 AND NOT STPINV1;
  //   INV_1_ON := _t1;
  //   RUN_1 := _t1;

// Rung 9: DAMPER 1 ON
  LD %S12                 (* SB_RUNMODE *)
  MPS
  AND( %M5                (* S_LOCAL_1 *)
  AND %M62                (* FLAG_MAN_DMPR1 *)
  OR( %M4                 (* S_REMOTE_1 *)
  AND( %M62               (* FLAG_MAN_DMPR1 *)
  ANDN %M100              (* MANUAL_AUTO_1 *)
  OR( %M82                (* FLAG_AUTO_DMPR_1 *)
  AND %M100               (* MANUAL_AUTO_1 *)
  )
  )
  )
  )
  ST %M103                (* DMPR_1_ON *)
  MPP
  [ %MW380 := %QW4.3 ]    (* DMPR_1_VIEW, AO_DMPR_1 *)
  // as ST:
  //   DMPR_1_ON := SB_RUNMODE AND (S_LOCAL_1 AND FLAG_MAN_DMPR1 OR S_REMOTE_1 AND (FLAG_MAN_DMPR1 AND NOT MANUAL_AUTO_1 OR FLAG_AUTO_DMPR_1 AND MANUAL_AUTO_1));
  //   IF SB_RUNMODE THEN DMPR_1_VIEW := AO_DMPR_1; END_IF;

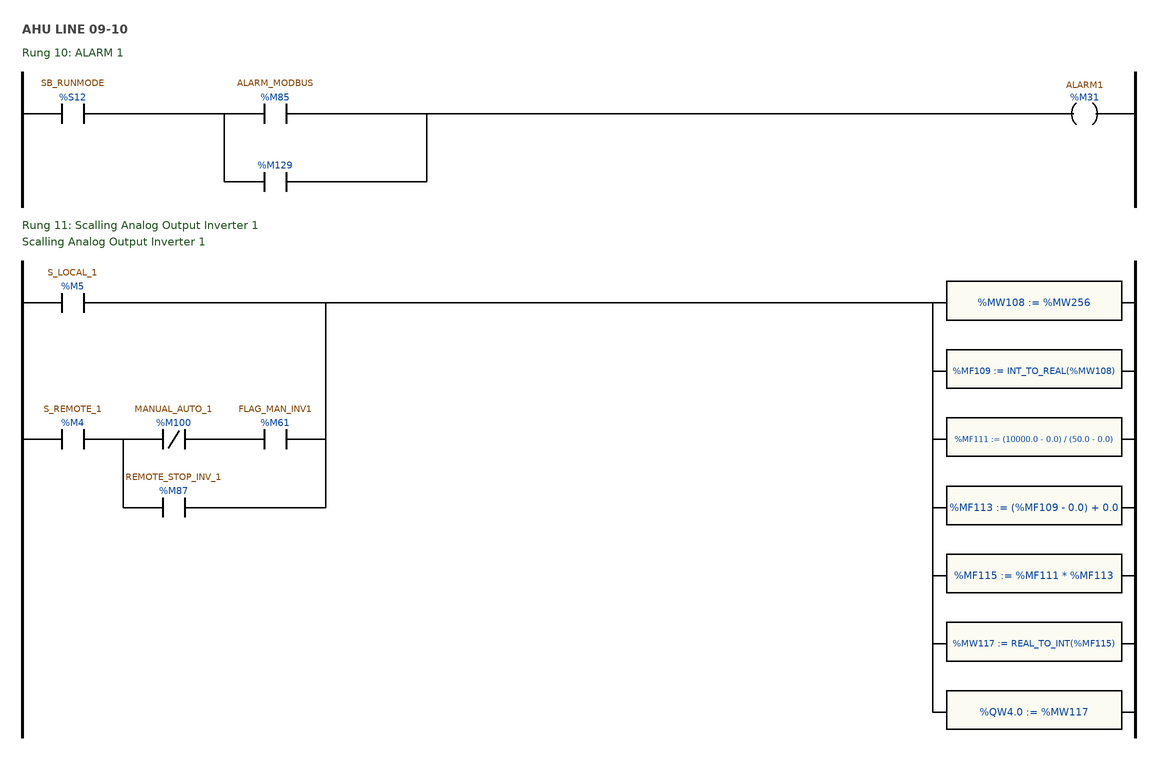

// Rung 10: ALARM 1
  LD %S12                 (* SB_RUNMODE *)
  AND( %M85               (* ALARM_MODBUS *)
  OR %M129
  )
  ST %M31                 (* ALARM1 *)
  // as ST:
  //   ALARM1 := SB_RUNMODE AND (ALARM_MODBUS OR %M129);

// Rung 11: Scalling Analog Output Inverter 1
// Scalling Analog Output Inverter 1
  LD %M5                  (* S_LOCAL_1 *)
  OR( %M4                 (* S_REMOTE_1 *)
  AND(N %M100             (* MANUAL_AUTO_1 *)
  AND %M61                (* FLAG_MAN_INV1 *)
  OR %M87                 (* REMOTE_STOP_INV_1 *)
  )
  )
  [ %MW108 := %MW256 ]    (* SET_SPEED_INV_1 *)
  [ %MF109 := INT_TO_REAL ( %MW108 ) ]
  [%MF111 := (10000.0 - 0.0) / (50.0 - 0.0)]
  [%MF113 := (%MF109 - 0.0) + 0.0]
  [ %MF115 := %MF111 * %MF113 ]
  [ %MW117 := REAL_TO_INT ( %MF115 ) ](* AO_SCALE_TEMP_1 *)
  [ %QW4.0 := %MW117 ]    (* AO_INV_1, AO_SCALE_TEMP_1 *)
  // as ST:
  //   IF S_LOCAL_1 OR S_REMOTE_1 AND (NOT MANUAL_AUTO_1 AND FLAG_MAN_INV1 OR REMOTE_STOP_INV_1) THEN %MW108 := SET_SPEED_INV_1; END_IF;
  //   IF S_LOCAL_1 OR S_REMOTE_1 AND (NOT MANUAL_AUTO_1 AND FLAG_MAN_INV1 OR REMOTE_STOP_INV_1) THEN %MF109 := INT_TO_REAL ( %MW108 ); END_IF;
  //   IF S_LOCAL_1 OR S_REMOTE_1 AND (NOT MANUAL_AUTO_1 AND FLAG_MAN_INV1 OR REMOTE_STOP_INV_1) THEN %MF111 := (10000.0 - 0.0) / (50.0 - 0.0); END_IF;
  //   IF S_LOCAL_1 OR S_REMOTE_1 AND (NOT MANUAL_AUTO_1 AND FLAG_MAN_INV1 OR REMOTE_STOP_INV_1) THEN %MF113 := (%MF109 - 0.0) + 0.0; END_IF;
  //   IF S_LOCAL_1 OR S_REMOTE_1 AND (NOT MANUAL_AUTO_1 AND FLAG_MAN_INV1 OR REMOTE_STOP_INV_1) THEN %MF115 := %MF111 * %MF113; END_IF;
  //   IF S_LOCAL_1 OR S_REMOTE_1 AND (NOT MANUAL_AUTO_1 AND FLAG_MAN_INV1 OR REMOTE_STOP_INV_1) THEN AO_SCALE_TEMP_1 := REAL_TO_INT ( %MF115 ); END_IF;
  //   IF S_LOCAL_1 OR S_REMOTE_1 AND (NOT MANUAL_AUTO_1 AND FLAG_MAN_INV1 OR REMOTE_STOP_INV_1) THEN AO_INV_1 := AO_SCALE_TEMP_1; END_IF;

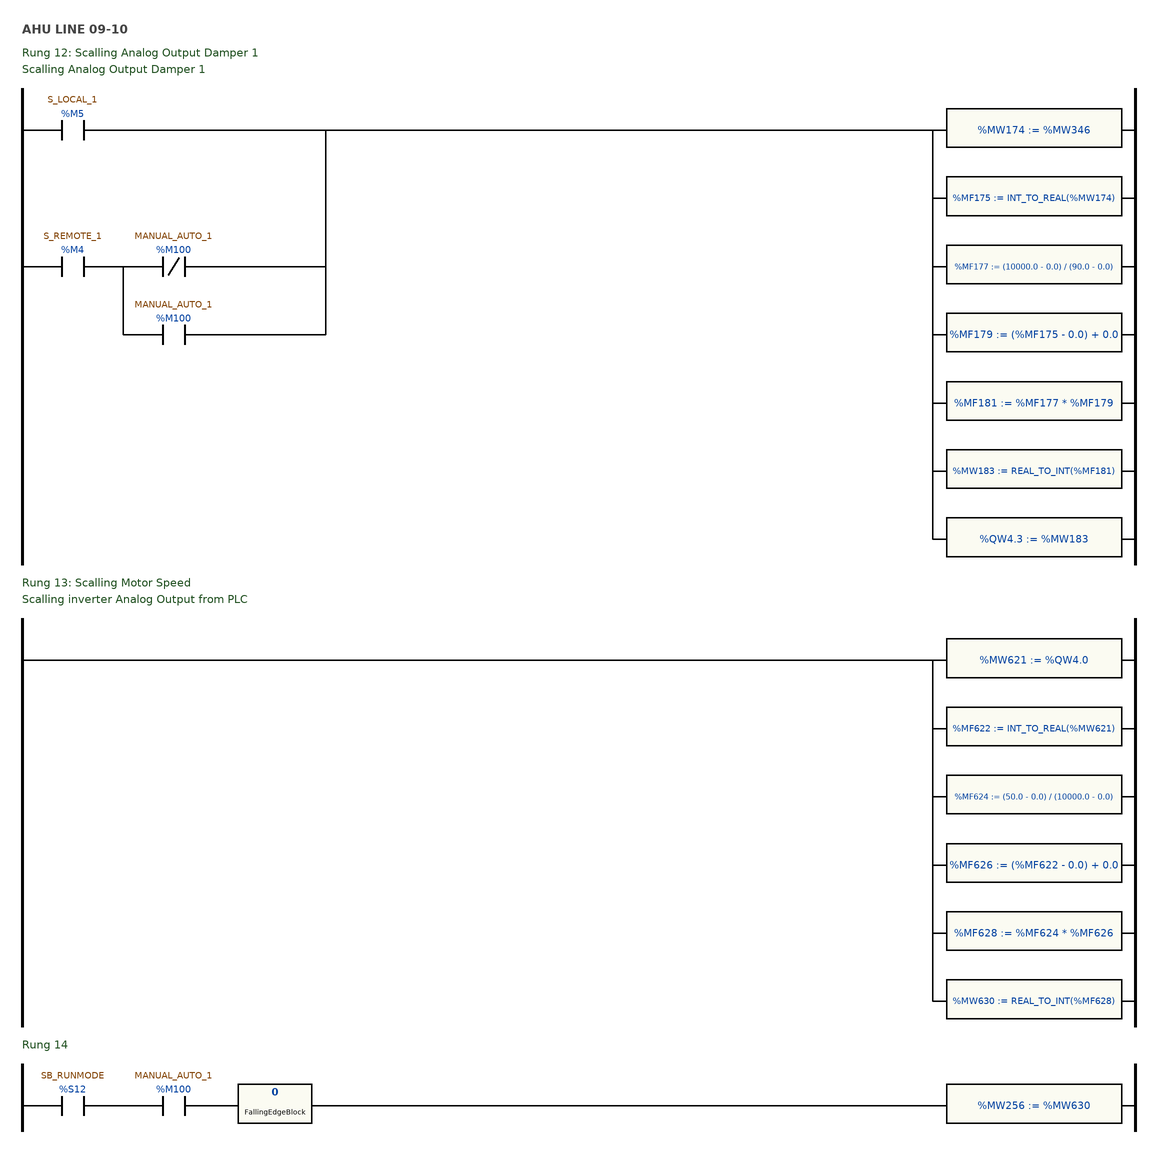

// Rung 12: Scalling Analog Output Damper 1
// Scalling Analog Output Damper 1
  LD %M5                  (* S_LOCAL_1 *)
  OR( %M4                 (* S_REMOTE_1 *)
  AND(N %M100             (* MANUAL_AUTO_1 *)
  OR %M100                (* MANUAL_AUTO_1 *)
  )
  )
  [ %MW174 := %MW346 ]    (* SET_DAMPER_POSITION_1 *)
  [ %MF175 := INT_TO_REAL ( %MW174 ) ]
  [%MF177 := (10000.0 - 0.0) / (90.0 - 0.0)]
  [%MF179 := (%MF175 - 0.0) + 0.0]
  [ %MF181 := %MF177 * %MF179 ]
  [ %MW183 := REAL_TO_INT ( %MF181 ) ](* AO_SCALE_HUMIDITY_1 *)
  [ %QW4.3 := %MW183 ]    (* AO_DMPR_1, AO_SCALE_HUMIDITY_1 *)
  // as ST:
  //   IF S_LOCAL_1 OR S_REMOTE_1 AND (NOT MANUAL_AUTO_1 OR MANUAL_AUTO_1) THEN %MW174 := SET_DAMPER_POSITION_1; END_IF;
  //   IF S_LOCAL_1 OR S_REMOTE_1 AND (NOT MANUAL_AUTO_1 OR MANUAL_AUTO_1) THEN %MF175 := INT_TO_REAL ( %MW174 ); END_IF;
  //   IF S_LOCAL_1 OR S_REMOTE_1 AND (NOT MANUAL_AUTO_1 OR MANUAL_AUTO_1) THEN %MF177 := (10000.0 - 0.0) / (90.0 - 0.0); END_IF;
  //   IF S_LOCAL_1 OR S_REMOTE_1 AND (NOT MANUAL_AUTO_1 OR MANUAL_AUTO_1) THEN %MF179 := (%MF175 - 0.0) + 0.0; END_IF;
  //   IF S_LOCAL_1 OR S_REMOTE_1 AND (NOT MANUAL_AUTO_1 OR MANUAL_AUTO_1) THEN %MF181 := %MF177 * %MF179; END_IF;
  //   IF S_LOCAL_1 OR S_REMOTE_1 AND (NOT MANUAL_AUTO_1 OR MANUAL_AUTO_1) THEN AO_SCALE_HUMIDITY_1 := REAL_TO_INT ( %MF181 ); END_IF;
  //   IF S_LOCAL_1 OR S_REMOTE_1 AND (NOT MANUAL_AUTO_1 OR MANUAL_AUTO_1) THEN AO_DMPR_1 := AO_SCALE_HUMIDITY_1; END_IF;

// Rung 13: Scalling Motor Speed
// Scalling inverter Analog Output from PLC
  LD 1
  [ %MW621 := %QW4.0 ]    (* AO_INV_1 *)
  [ %MF622 := INT_TO_REAL ( %MW621 ) ]
  [%MF624 := (50.0 - 0.0) / (10000.0 - 0.0)]
  [%MF626 := (%MF622 - 0.0) + 0.0]
  [ %MF628 := %MF624 * %MF626 ]
  [ %MW630 := REAL_TO_INT ( %MF628 ) ](* INV_1_HZ *)
  // as ST:
  //   %MW621 := AO_INV_1;
  //   %MF622 := INT_TO_REAL ( %MW621 );
  //   %MF624 := (50.0 - 0.0) / (10000.0 - 0.0);
  //   %MF626 := (%MF622 - 0.0) + 0.0;
  //   %MF628 := %MF624 * %MF626;
  //   INV_1_HZ := REAL_TO_INT ( %MF628 );

// Rung 14
  LD %S12                 (* SB_RUNMODE *)
  AND %M100               (* MANUAL_AUTO_1 *)
  FALLING0
  [ %MW256 := %MW630 ]    (* SET_SPEED_INV_1, INV_1_HZ *)
  // as ST:
  //   IF FALLING(SB_RUNMODE AND MANUAL_AUTO_1) THEN SET_SPEED_INV_1 := INV_1_HZ; END_IF;

POU AHU LINE 11-12
  (* SectionNumber=3 *)

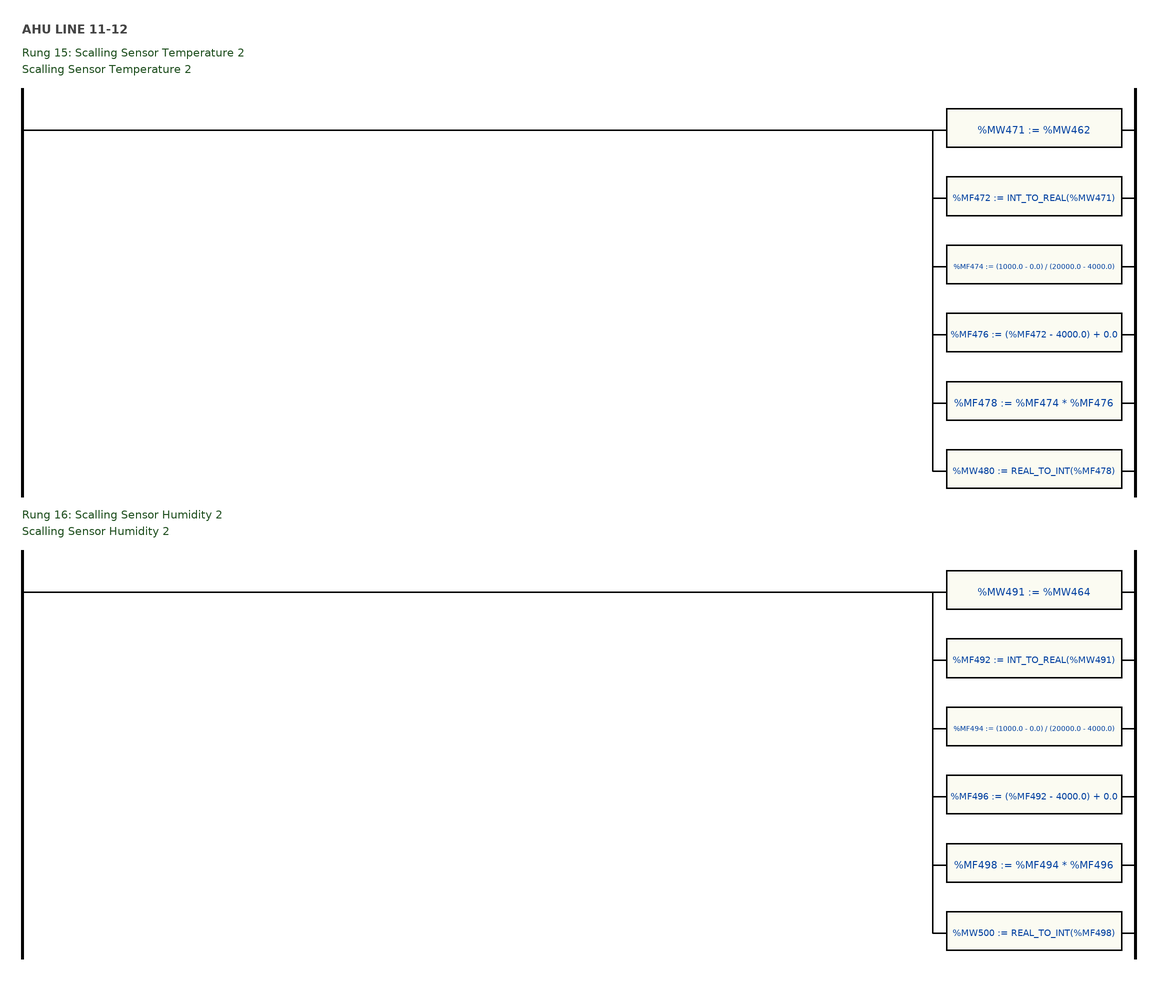

// Rung 15: Scalling Sensor Temperature 2
// Scalling Sensor Temperature 2
  LD 1
  [ %MW471 := %MW462 ]    (* TEMP_2_DATA_SERIAL *)
  [ %MF472 := INT_TO_REAL ( %MW471 ) ]
  [%MF474 := (1000.0 - 0.0) / (20000.0 - 4000.0)]
  [%MF476 := (%MF472 - 4000.0) + 0.0]
  [ %MF478 := %MF474 * %MF476 ]
  [ %MW480 := REAL_TO_INT ( %MF478 ) ](* AI_SCALE_TEMP_2 *)
  // as ST:
  //   %MW471 := TEMP_2_DATA_SERIAL;
  //   %MF472 := INT_TO_REAL ( %MW471 );
  //   %MF474 := (1000.0 - 0.0) / (20000.0 - 4000.0);
  //   %MF476 := (%MF472 - 4000.0) + 0.0;
  //   %MF478 := %MF474 * %MF476;
  //   AI_SCALE_TEMP_2 := REAL_TO_INT ( %MF478 );

// Rung 16: Scalling Sensor Humidity 2
// Scalling Sensor Humidity 2
  LD 1
  [ %MW491 := %MW464 ]    (* HUMIDITY_2_DATA_SERIAL *)
  [ %MF492 := INT_TO_REAL ( %MW491 ) ]
  [%MF494 := (1000.0 - 0.0) / (20000.0 - 4000.0)]
  [%MF496 := (%MF492 - 4000.0) + 0.0]
  [ %MF498 := %MF494 * %MF496 ]
  [ %MW500 := REAL_TO_INT ( %MF498 ) ](* AI_SCALE_HUMIDITY_2 *)
  // as ST:
  //   %MW491 := HUMIDITY_2_DATA_SERIAL;
  //   %MF492 := INT_TO_REAL ( %MW491 );
  //   %MF494 := (1000.0 - 0.0) / (20000.0 - 4000.0);
  //   %MF496 := (%MF492 - 4000.0) + 0.0;
  //   %MF498 := %MF494 * %MF496;
  //   AI_SCALE_HUMIDITY_2 := REAL_TO_INT ( %MF498 );

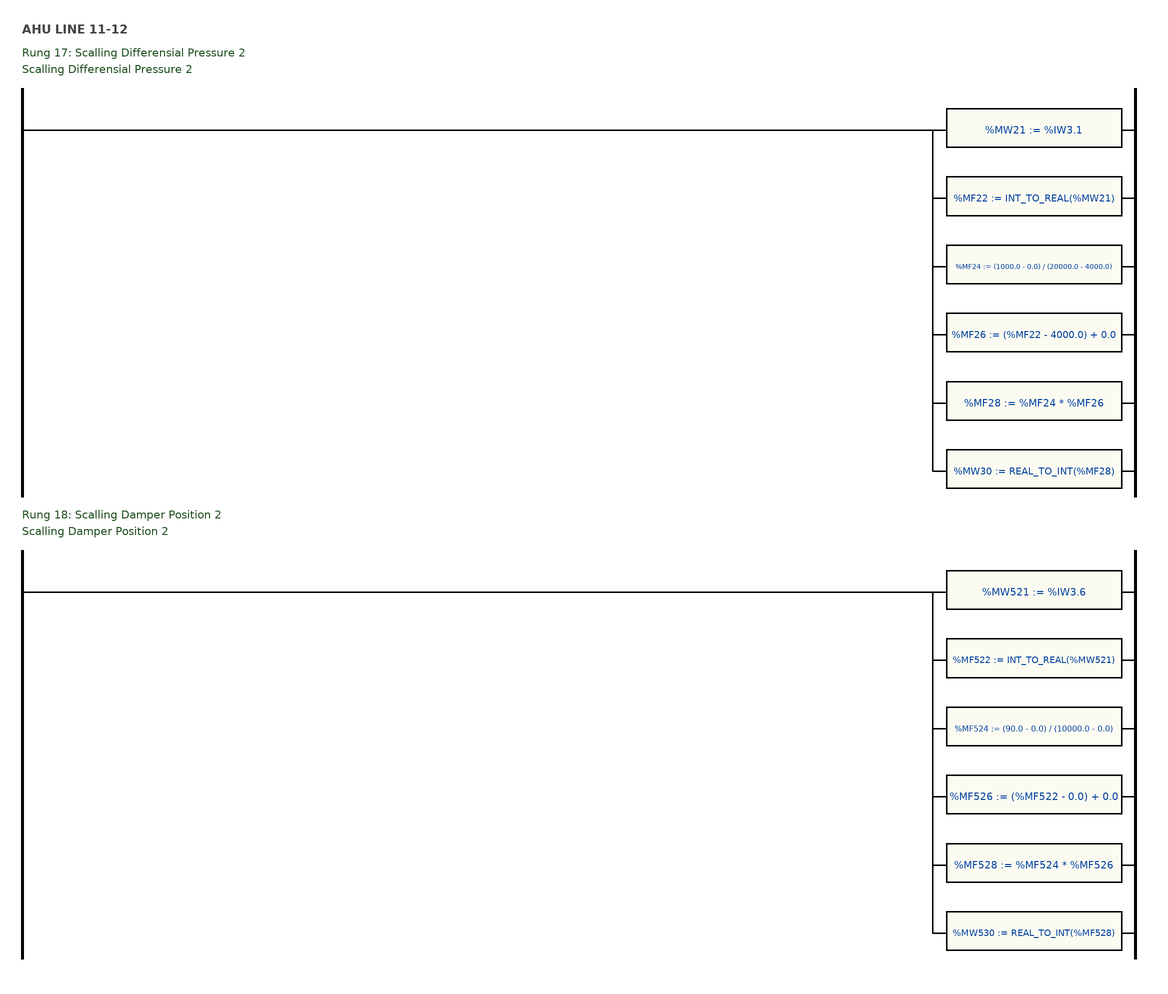

// Rung 17: Scalling Differensial Pressure 2
// Scalling Differensial Pressure 2
  LD 1
  [ %MW21 := %IW3.1 ]     (* PRESS_AHU_2 *)
  [ %MF22 := INT_TO_REAL ( %MW21 ) ]
  [%MF24 := (1000.0 - 0.0) / (20000.0 - 4000.0)]
  [%MF26 := (%MF22 - 4000.0) + 0.0]
  [ %MF28 := %MF24 * %MF26 ]
  [ %MW30 := REAL_TO_INT ( %MF28 ) ](* AI_SCALE_DIFF_PRESSURE_2 *)
  // as ST:
  //   %MW21 := PRESS_AHU_2;
  //   %MF22 := INT_TO_REAL ( %MW21 );
  //   %MF24 := (1000.0 - 0.0) / (20000.0 - 4000.0);
  //   %MF26 := (%MF22 - 4000.0) + 0.0;
  //   %MF28 := %MF24 * %MF26;
  //   AI_SCALE_DIFF_PRESSURE_2 := REAL_TO_INT ( %MF28 );

// Rung 18: Scalling Damper Position 2
// Scalling Damper Position 2
  LD 1
  [ %MW521 := %IW3.6 ]    (* DAMP_POS_AHU_2 *)
  [ %MF522 := INT_TO_REAL ( %MW521 ) ]
  [%MF524 := (90.0 - 0.0) / (10000.0 - 0.0)]
  [%MF526 := (%MF522 - 0.0) + 0.0]
  [ %MF528 := %MF524 * %MF526 ]
  [ %MW530 := REAL_TO_INT ( %MF528 ) ](* AI_SCALE_DAMPER_POSITION_2 *)
  // as ST:
  //   %MW521 := DAMP_POS_AHU_2;
  //   %MF522 := INT_TO_REAL ( %MW521 );
  //   %MF524 := (90.0 - 0.0) / (10000.0 - 0.0);
  //   %MF526 := (%MF522 - 0.0) + 0.0;
  //   %MF528 := %MF524 * %MF526;
  //   AI_SCALE_DAMPER_POSITION_2 := REAL_TO_INT ( %MF528 );

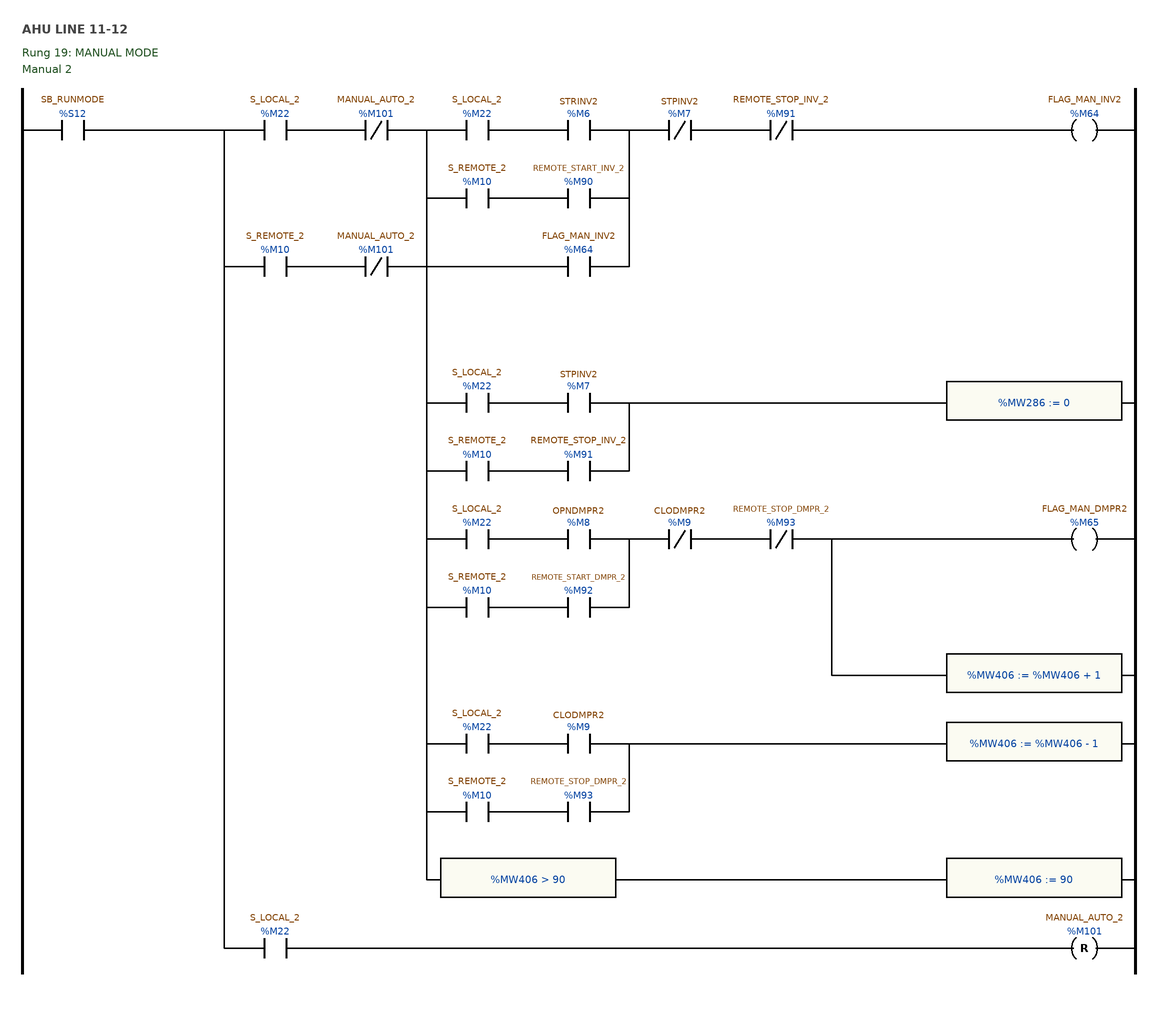

// Rung 19: MANUAL MODE
// Manual 2
  LD %S12                 (* SB_RUNMODE *)
  MPS
  AND( %M22               (* S_LOCAL_2 *)
  ANDN %M101              (* MANUAL_AUTO_2 *)
  OR( %M10                (* S_REMOTE_2 *)
  ANDN %M101              (* MANUAL_AUTO_2 *)
  )
  )
  MPS
  AND( %M22               (* S_LOCAL_2 *)
  AND %M6                 (* STRINV2 *)
  OR( %M10                (* S_REMOTE_2 *)
  AND %M90                (* REMOTE_START_INV_2 *)
  )
  OR %M64                 (* FLAG_MAN_INV2 *)
  )
  ANDN %M7                (* STPINV2 *)
  ANDN %M91               (* REMOTE_STOP_INV_2 *)
  ST %M64                 (* FLAG_MAN_INV2 *)
  MRD
  AND( %M22               (* S_LOCAL_2 *)
  AND %M7                 (* STPINV2 *)
  OR( %M10                (* S_REMOTE_2 *)
  AND %M91                (* REMOTE_STOP_INV_2 *)
  )
  )
  [ %MW286 := 0 ]         (* SET_SPEED_INV_2 *)
  MRD
  AND( %M22               (* S_LOCAL_2 *)
  AND %M8                 (* OPNDMPR2 *)
  OR( %M10                (* S_REMOTE_2 *)
  AND %M92                (* REMOTE_START_DMPR_2 *)
  )
  )
  ANDN %M9                (* CLODMPR2 *)
  ANDN %M93               (* REMOTE_STOP_DMPR_2 *)
  ST %M65                 (* FLAG_MAN_DMPR2 *)
  [ %MW406 := %MW406 + 1 ](* SET_DAMPER_2_POSITION, SET_DAMPER_2_POSITION *)
  MRD
  AND( %M22               (* S_LOCAL_2 *)
  AND %M9                 (* CLODMPR2 *)
  OR( %M10                (* S_REMOTE_2 *)
  AND %M93                (* REMOTE_STOP_DMPR_2 *)
  )
  )
  [ %MW406 := %MW406 - 1 ](* SET_DAMPER_2_POSITION, SET_DAMPER_2_POSITION *)
  MPP
  AND [ %MW406 > 90 ]     (* SET_DAMPER_2_POSITION *)
  [ %MW406 := 90 ]        (* SET_DAMPER_2_POSITION *)
  MPP
  AND %M22                (* S_LOCAL_2 *)
  R %M101                 (* MANUAL_AUTO_2 *)
  // as ST:
  //   FLAG_MAN_INV2 := SB_RUNMODE AND (S_LOCAL_2 AND NOT MANUAL_AUTO_2 OR S_REMOTE_2 AND NOT MANUAL_AUTO_2) AND (S_LOCAL_2 AND STRINV2 OR S_REMOTE_2 AND REMOTE_START_INV_2 OR FLAG_MAN_INV2) AND NOT STPINV2 AND NOT REMOTE_STOP_INV_2;
  //   IF SB_RUNMODE AND (S_LOCAL_2 AND NOT MANUAL_AUTO_2 OR S_REMOTE_2 AND NOT MANUAL_AUTO_2) AND (S_LOCAL_2 AND STPINV2 OR S_REMOTE_2 AND REMOTE_STOP_INV_2) THEN SET_SPEED_INV_2 := 0; END_IF;
  //   FLAG_MAN_DMPR2 := SB_RUNMODE AND (S_LOCAL_2 AND NOT MANUAL_AUTO_2 OR S_REMOTE_2 AND NOT MANUAL_AUTO_2) AND (S_LOCAL_2 AND OPNDMPR2 OR S_REMOTE_2 AND REMOTE_START_DMPR_2) AND NOT CLODMPR2 AND NOT REMOTE_STOP_DMPR_2;
  //   IF SB_RUNMODE AND (S_LOCAL_2 AND NOT MANUAL_AUTO_2 OR S_REMOTE_2 AND NOT MANUAL_AUTO_2) AND (S_LOCAL_2 AND OPNDMPR2 OR S_REMOTE_2 AND REMOTE_START_DMPR_2) AND NOT CLODMPR2 AND NOT REMOTE_STOP_DMPR_2 THEN SET_DAMPER_2_POSITION := SET_DAMPER_2_POSITION + 1; END_IF;
  //   IF SB_RUNMODE AND (S_LOCAL_2 AND NOT MANUAL_AUTO_2 OR S_REMOTE_2 AND NOT MANUAL_AUTO_2) AND (S_LOCAL_2 AND CLODMPR2 OR S_REMOTE_2 AND REMOTE_STOP_DMPR_2) THEN SET_DAMPER_2_POSITION := SET_DAMPER_2_POSITION - 1; END_IF;
  //   IF SB_RUNMODE AND (S_LOCAL_2 AND NOT MANUAL_AUTO_2 OR S_REMOTE_2 AND NOT MANUAL_AUTO_2) AND SET_DAMPER_2_POSITION > 90 THEN SET_DAMPER_2_POSITION := 90; END_IF;
  //   IF SB_RUNMODE AND S_LOCAL_2 THEN MANUAL_AUTO_2 := FALSE; END_IF;

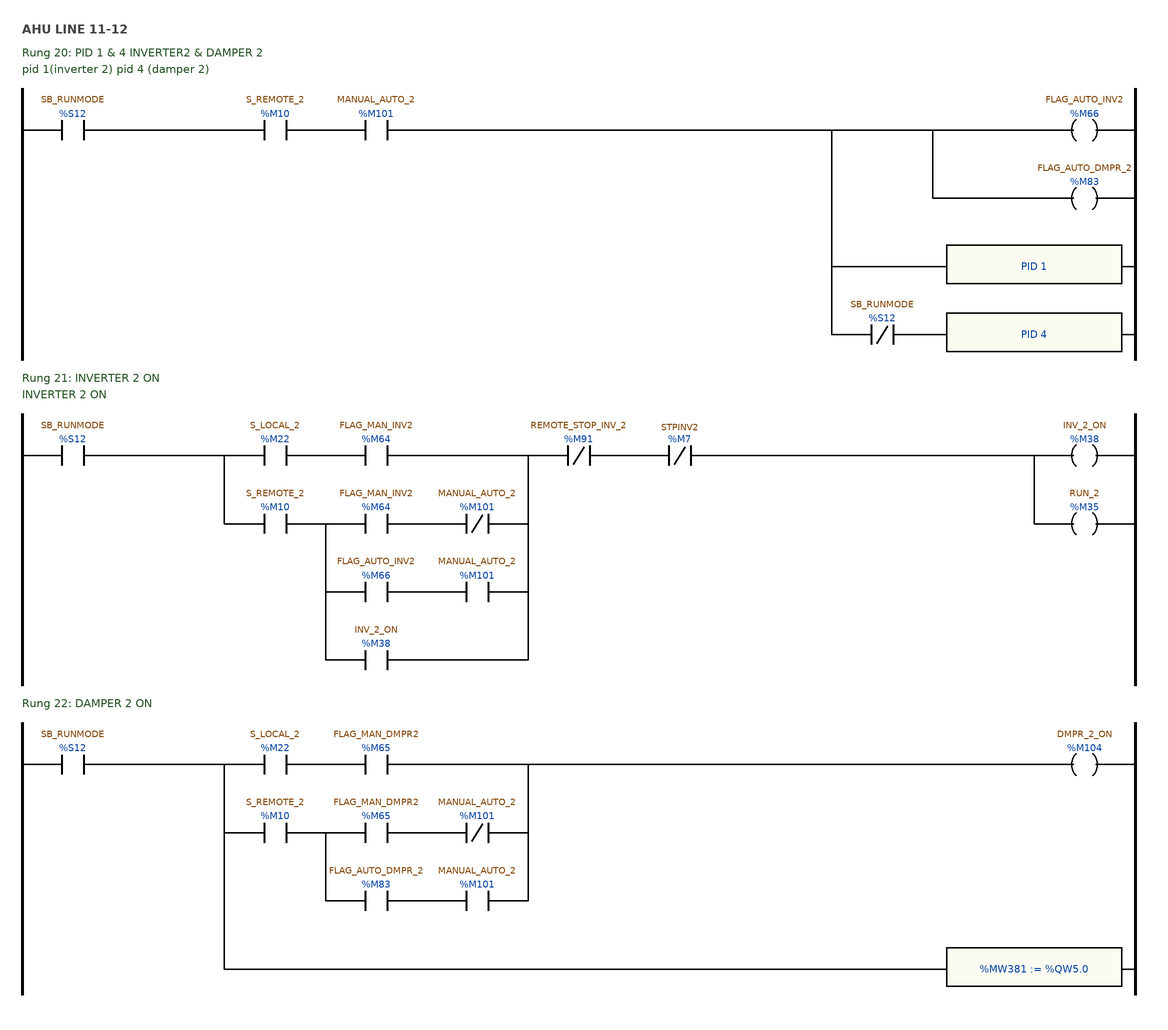

// Rung 20: PID 1 & 4 INVERTER2 & DAMPER 2
// pid 1(inverter 2) pid 4 (damper 2)
  LD %S12                 (* SB_RUNMODE *)
  AND %M10                (* S_REMOTE_2 *)
  AND %M101               (* MANUAL_AUTO_2 *)
  MPS
  ST %M66                 (* FLAG_AUTO_INV2 *)
  ST %M83                 (* FLAG_AUTO_DMPR_2 *)
  MRD
  [ PID 1 ]
  MPP
  ANDN %S12               (* SB_RUNMODE *)
  [ PID 4 ]
  // as ST:
  //   FLAG_AUTO_INV2 := SB_RUNMODE AND S_REMOTE_2 AND MANUAL_AUTO_2;
  //   FLAG_AUTO_DMPR_2 := SB_RUNMODE AND S_REMOTE_2 AND MANUAL_AUTO_2;
  //   IF SB_RUNMODE AND S_REMOTE_2 AND MANUAL_AUTO_2 THEN PID 1; END_IF;
  //   IF SB_RUNMODE AND S_REMOTE_2 AND MANUAL_AUTO_2 AND NOT SB_RUNMODE THEN PID 4; END_IF;

// Rung 21: INVERTER 2 ON
// INVERTER 2 ON
  LD %S12                 (* SB_RUNMODE *)
  AND( %M22               (* S_LOCAL_2 *)
  AND %M64                (* FLAG_MAN_INV2 *)
  OR( %M10                (* S_REMOTE_2 *)
  AND( %M64               (* FLAG_MAN_INV2 *)
  ANDN %M101              (* MANUAL_AUTO_2 *)
  OR( %M66                (* FLAG_AUTO_INV2 *)
  AND %M101               (* MANUAL_AUTO_2 *)
  )
  OR %M38                 (* INV_2_ON *)
  )
  )
  )
  ANDN %M91               (* REMOTE_STOP_INV_2 *)
  ANDN %M7                (* STPINV2 *)
  ST %M38                 (* INV_2_ON *)
  ST %M35                 (* RUN_2 *)
  // as ST:
  //   _t1 := SB_RUNMODE AND (S_LOCAL_2 AND FLAG_MAN_INV2 OR S_REMOTE_2 AND (FLAG_MAN_INV2 AND NOT MANUAL_AUTO_2 OR FLAG_AUTO_INV2 AND MANUAL_AUTO_2 OR INV_2_ON)) AND NOT REMOTE_STOP_INV_2 AND NOT STPINV2;
  //   INV_2_ON := _t1;
  //   RUN_2 := _t1;

// Rung 22: DAMPER 2 ON
  LD %S12                 (* SB_RUNMODE *)
  MPS
  AND( %M22               (* S_LOCAL_2 *)
  AND %M65                (* FLAG_MAN_DMPR2 *)
  OR( %M10                (* S_REMOTE_2 *)
  AND( %M65               (* FLAG_MAN_DMPR2 *)
  ANDN %M101              (* MANUAL_AUTO_2 *)
  OR( %M83                (* FLAG_AUTO_DMPR_2 *)
  AND %M101               (* MANUAL_AUTO_2 *)
  )
  )
  )
  )
  ST %M104                (* DMPR_2_ON *)
  MPP
  [ %MW381 := %QW5.0 ]    (* DMPR_2_VIEW, AO_DMPR_2 *)
  // as ST:
  //   DMPR_2_ON := SB_RUNMODE AND (S_LOCAL_2 AND FLAG_MAN_DMPR2 OR S_REMOTE_2 AND (FLAG_MAN_DMPR2 AND NOT MANUAL_AUTO_2 OR FLAG_AUTO_DMPR_2 AND MANUAL_AUTO_2));
  //   IF SB_RUNMODE THEN DMPR_2_VIEW := AO_DMPR_2; END_IF;

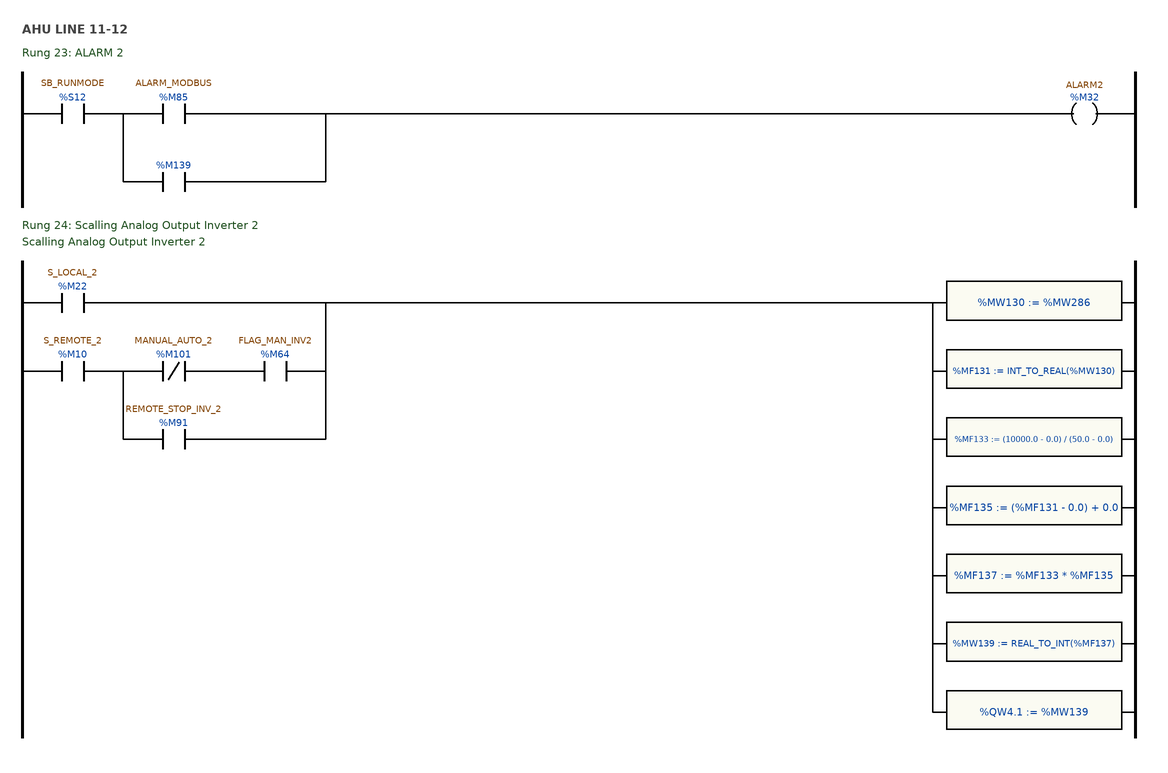

// Rung 23: ALARM 2
  LD %S12                 (* SB_RUNMODE *)
  AND( %M85               (* ALARM_MODBUS *)
  OR %M139
  )
  ST %M32                 (* ALARM2 *)
  // as ST:
  //   ALARM2 := SB_RUNMODE AND (ALARM_MODBUS OR %M139);

// Rung 24: Scalling Analog Output Inverter 2
// Scalling Analog Output Inverter 2
  LD %M22                 (* S_LOCAL_2 *)
  OR( %M10                (* S_REMOTE_2 *)
  AND(N %M101             (* MANUAL_AUTO_2 *)
  AND %M64                (* FLAG_MAN_INV2 *)
  OR %M91                 (* REMOTE_STOP_INV_2 *)
  )
  )
  [ %MW130 := %MW286 ]    (* SET_SPEED_INV_2 *)
  [ %MF131 := INT_TO_REAL ( %MW130 ) ]
  [%MF133 := (10000.0 - 0.0) / (50.0 - 0.0)]
  [%MF135 := (%MF131 - 0.0) + 0.0]
  [ %MF137 := %MF133 * %MF135 ]
  [ %MW139 := REAL_TO_INT ( %MF137 ) ](* AO_SCALE_TEMP_2 *)
  [ %QW4.1 := %MW139 ]    (* AO_INV_2, AO_SCALE_TEMP_2 *)
  // as ST:
  //   IF S_LOCAL_2 OR S_REMOTE_2 AND (NOT MANUAL_AUTO_2 AND FLAG_MAN_INV2 OR REMOTE_STOP_INV_2) THEN %MW130 := SET_SPEED_INV_2; END_IF;
  //   IF S_LOCAL_2 OR S_REMOTE_2 AND (NOT MANUAL_AUTO_2 AND FLAG_MAN_INV2 OR REMOTE_STOP_INV_2) THEN %MF131 := INT_TO_REAL ( %MW130 ); END_IF;
  //   IF S_LOCAL_2 OR S_REMOTE_2 AND (NOT MANUAL_AUTO_2 AND FLAG_MAN_INV2 OR REMOTE_STOP_INV_2) THEN %MF133 := (10000.0 - 0.0) / (50.0 - 0.0); END_IF;
  //   IF S_LOCAL_2 OR S_REMOTE_2 AND (NOT MANUAL_AUTO_2 AND FLAG_MAN_INV2 OR REMOTE_STOP_INV_2) THEN %MF135 := (%MF131 - 0.0) + 0.0; END_IF;
  //   IF S_LOCAL_2 OR S_REMOTE_2 AND (NOT MANUAL_AUTO_2 AND FLAG_MAN_INV2 OR REMOTE_STOP_INV_2) THEN %MF137 := %MF133 * %MF135; END_IF;
  //   IF S_LOCAL_2 OR S_REMOTE_2 AND (NOT MANUAL_AUTO_2 AND FLAG_MAN_INV2 OR REMOTE_STOP_INV_2) THEN AO_SCALE_TEMP_2 := REAL_TO_INT ( %MF137 ); END_IF;
  //   IF S_LOCAL_2 OR S_REMOTE_2 AND (NOT MANUAL_AUTO_2 AND FLAG_MAN_INV2 OR REMOTE_STOP_INV_2) THEN AO_INV_2 := AO_SCALE_TEMP_2; END_IF;

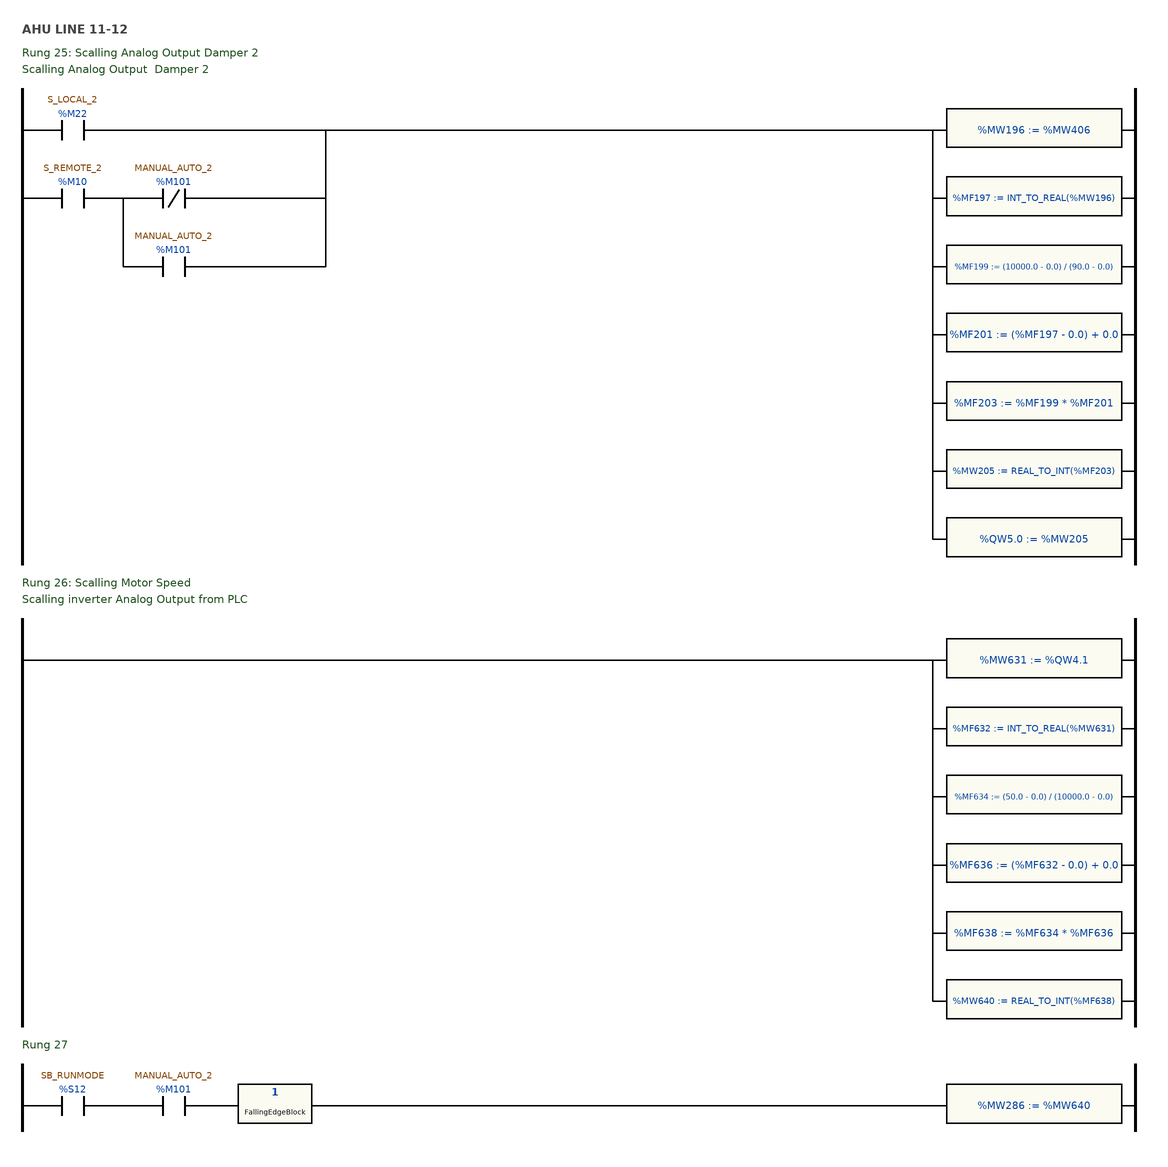

// Rung 25: Scalling Analog Output Damper 2
// Scalling Analog Output  Damper 2
  LD %M22                 (* S_LOCAL_2 *)
  OR( %M10                (* S_REMOTE_2 *)
  AND(N %M101             (* MANUAL_AUTO_2 *)
  OR %M101                (* MANUAL_AUTO_2 *)
  )
  )
  [ %MW196 := %MW406 ]    (* SET_DAMPER_2_POSITION *)
  [ %MF197 := INT_TO_REAL ( %MW196 ) ]
  [%MF199 := (10000.0 - 0.0) / (90.0 - 0.0)]
  [%MF201 := (%MF197 - 0.0) + 0.0]
  [ %MF203 := %MF199 * %MF201 ]
  [ %MW205 := REAL_TO_INT ( %MF203 ) ](* AO_SCALE_HUMIDITY_2 *)
  [ %QW5.0 := %MW205 ]    (* AO_DMPR_2, AO_SCALE_HUMIDITY_2 *)
  // as ST:
  //   IF S_LOCAL_2 OR S_REMOTE_2 AND (NOT MANUAL_AUTO_2 OR MANUAL_AUTO_2) THEN %MW196 := SET_DAMPER_2_POSITION; END_IF;
  //   IF S_LOCAL_2 OR S_REMOTE_2 AND (NOT MANUAL_AUTO_2 OR MANUAL_AUTO_2) THEN %MF197 := INT_TO_REAL ( %MW196 ); END_IF;
  //   IF S_LOCAL_2 OR S_REMOTE_2 AND (NOT MANUAL_AUTO_2 OR MANUAL_AUTO_2) THEN %MF199 := (10000.0 - 0.0) / (90.0 - 0.0); END_IF;
  //   IF S_LOCAL_2 OR S_REMOTE_2 AND (NOT MANUAL_AUTO_2 OR MANUAL_AUTO_2) THEN %MF201 := (%MF197 - 0.0) + 0.0; END_IF;
  //   IF S_LOCAL_2 OR S_REMOTE_2 AND (NOT MANUAL_AUTO_2 OR MANUAL_AUTO_2) THEN %MF203 := %MF199 * %MF201; END_IF;
  //   IF S_LOCAL_2 OR S_REMOTE_2 AND (NOT MANUAL_AUTO_2 OR MANUAL_AUTO_2) THEN AO_SCALE_HUMIDITY_2 := REAL_TO_INT ( %MF203 ); END_IF;
  //   IF S_LOCAL_2 OR S_REMOTE_2 AND (NOT MANUAL_AUTO_2 OR MANUAL_AUTO_2) THEN AO_DMPR_2 := AO_SCALE_HUMIDITY_2; END_IF;

// Rung 26: Scalling Motor Speed
// Scalling inverter Analog Output from PLC
  LD 1
  [ %MW631 := %QW4.1 ]    (* AO_INV_2 *)
  [ %MF632 := INT_TO_REAL ( %MW631 ) ]
  [%MF634 := (50.0 - 0.0) / (10000.0 - 0.0)]
  [%MF636 := (%MF632 - 0.0) + 0.0]
  [ %MF638 := %MF634 * %MF636 ]
  [ %MW640 := REAL_TO_INT ( %MF638 ) ](* INV_2_HZ *)
  // as ST:
  //   %MW631 := AO_INV_2;
  //   %MF632 := INT_TO_REAL ( %MW631 );
  //   %MF634 := (50.0 - 0.0) / (10000.0 - 0.0);
  //   %MF636 := (%MF632 - 0.0) + 0.0;
  //   %MF638 := %MF634 * %MF636;
  //   INV_2_HZ := REAL_TO_INT ( %MF638 );

// Rung 27
  LD %S12                 (* SB_RUNMODE *)
  AND %M101               (* MANUAL_AUTO_2 *)
  FALLING1
  [ %MW286 := %MW640 ]    (* SET_SPEED_INV_2, INV_2_HZ *)
  // as ST:
  //   IF FALLING(SB_RUNMODE AND MANUAL_AUTO_2) THEN SET_SPEED_INV_2 := INV_2_HZ; END_IF;

POU AHU LINE 17-18
  (* SectionNumber=4 *)

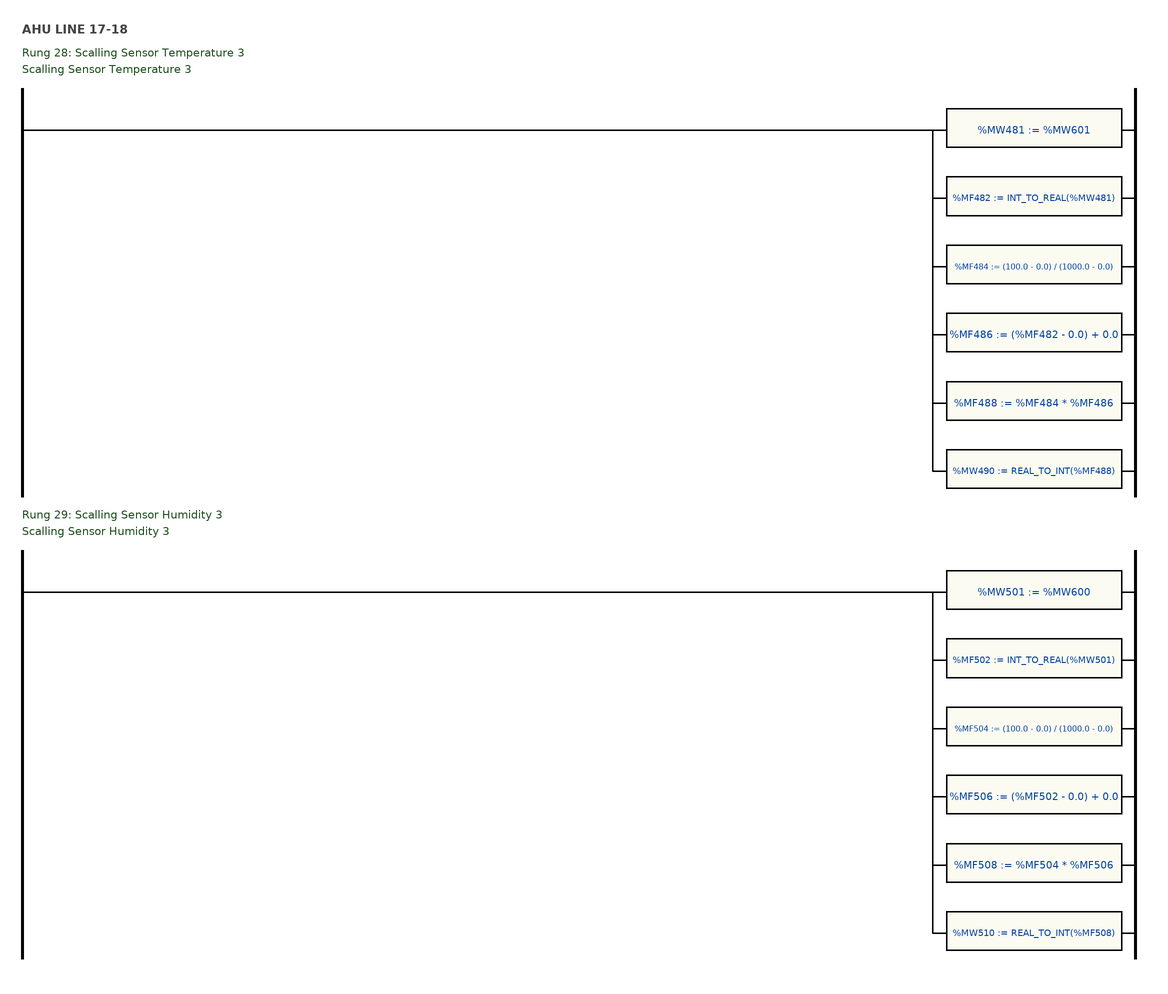

// Rung 28: Scalling Sensor Temperature 3
// Scalling Sensor Temperature 3
  LD 1
  [ %MW481 := %MW601 ]    (* TEMPERATURE_LINE_1718 *)
  [ %MF482 := INT_TO_REAL ( %MW481 ) ]
  [%MF484 := (100.0 - 0.0) / (1000.0 - 0.0)]
  [%MF486 := (%MF482 - 0.0) + 0.0]
  [ %MF488 := %MF484 * %MF486 ]
  [ %MW490 := REAL_TO_INT ( %MF488 ) ](* AI_SCALE_TEMP_3 *)
  // as ST:
  //   %MW481 := TEMPERATURE_LINE_1718;
  //   %MF482 := INT_TO_REAL ( %MW481 );
  //   %MF484 := (100.0 - 0.0) / (1000.0 - 0.0);
  //   %MF486 := (%MF482 - 0.0) + 0.0;
  //   %MF488 := %MF484 * %MF486;
  //   AI_SCALE_TEMP_3 := REAL_TO_INT ( %MF488 );

// Rung 29: Scalling Sensor Humidity 3
// Scalling Sensor Humidity 3
  LD 1
  [ %MW501 := %MW600 ]    (* HUMIDITY_LINE_1718 *)
  [ %MF502 := INT_TO_REAL ( %MW501 ) ]
  [%MF504 := (100.0 - 0.0) / (1000.0 - 0.0)]
  [%MF506 := (%MF502 - 0.0) + 0.0]
  [ %MF508 := %MF504 * %MF506 ]
  [ %MW510 := REAL_TO_INT ( %MF508 ) ](* AI_SCALE_HUMIDITY_3 *)
  // as ST:
  //   %MW501 := HUMIDITY_LINE_1718;
  //   %MF502 := INT_TO_REAL ( %MW501 );
  //   %MF504 := (100.0 - 0.0) / (1000.0 - 0.0);
  //   %MF506 := (%MF502 - 0.0) + 0.0;
  //   %MF508 := %MF504 * %MF506;
  //   AI_SCALE_HUMIDITY_3 := REAL_TO_INT ( %MF508 );

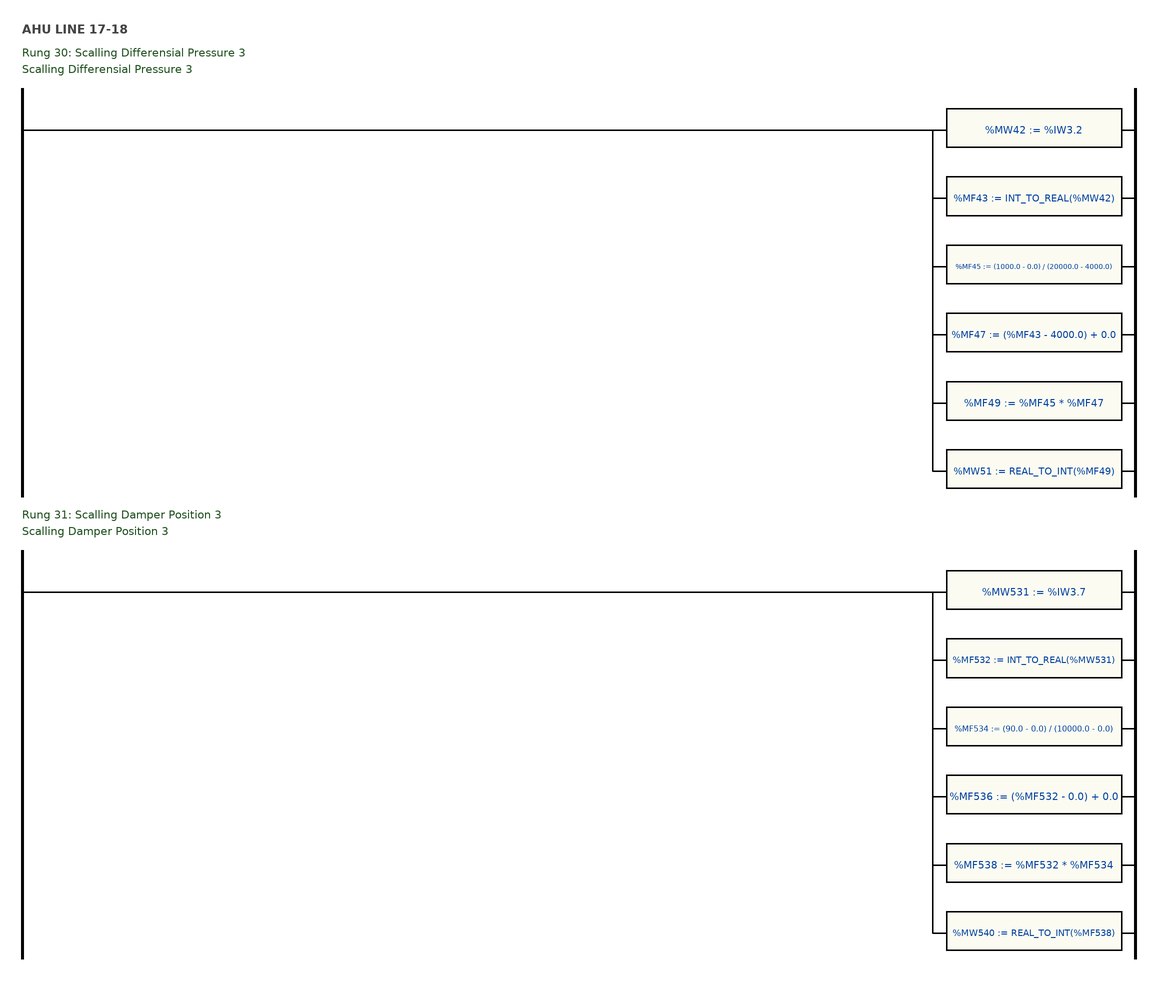

// Rung 30: Scalling Differensial Pressure 3
// Scalling Differensial Pressure 3
  LD 1
  [ %MW42 := %IW3.2 ]     (* PRESS_AHU_3 *)
  [ %MF43 := INT_TO_REAL ( %MW42 ) ]
  [%MF45 := (1000.0 - 0.0) / (20000.0 - 4000.0)]
  [%MF47 := (%MF43 - 4000.0) + 0.0]
  [ %MF49 := %MF45 * %MF47 ]
  [ %MW51 := REAL_TO_INT ( %MF49 ) ](* AI_SCALE_DIFF_PRESSURE_3 *)
  // as ST:
  //   %MW42 := PRESS_AHU_3;
  //   %MF43 := INT_TO_REAL ( %MW42 );
  //   %MF45 := (1000.0 - 0.0) / (20000.0 - 4000.0);
  //   %MF47 := (%MF43 - 4000.0) + 0.0;
  //   %MF49 := %MF45 * %MF47;
  //   AI_SCALE_DIFF_PRESSURE_3 := REAL_TO_INT ( %MF49 );

// Rung 31: Scalling Damper Position 3
// Scalling Damper Position 3
  LD 1
  [ %MW531 := %IW3.7 ]    (* DAMP_POS_AHU_3 *)
  [ %MF532 := INT_TO_REAL ( %MW531 ) ]
  [%MF534 := (90.0 - 0.0) / (10000.0 - 0.0)]
  [%MF536 := (%MF532 - 0.0) + 0.0]
  [ %MF538 := %MF532 * %MF534 ]
  [ %MW540 := REAL_TO_INT ( %MF538 ) ](* AI_SCALE_DAMPER_POSITION_3 *)
  // as ST:
  //   %MW531 := DAMP_POS_AHU_3;
  //   %MF532 := INT_TO_REAL ( %MW531 );
  //   %MF534 := (90.0 - 0.0) / (10000.0 - 0.0);
  //   %MF536 := (%MF532 - 0.0) + 0.0;
  //   %MF538 := %MF532 * %MF534;
  //   AI_SCALE_DAMPER_POSITION_3 := REAL_TO_INT ( %MF538 );

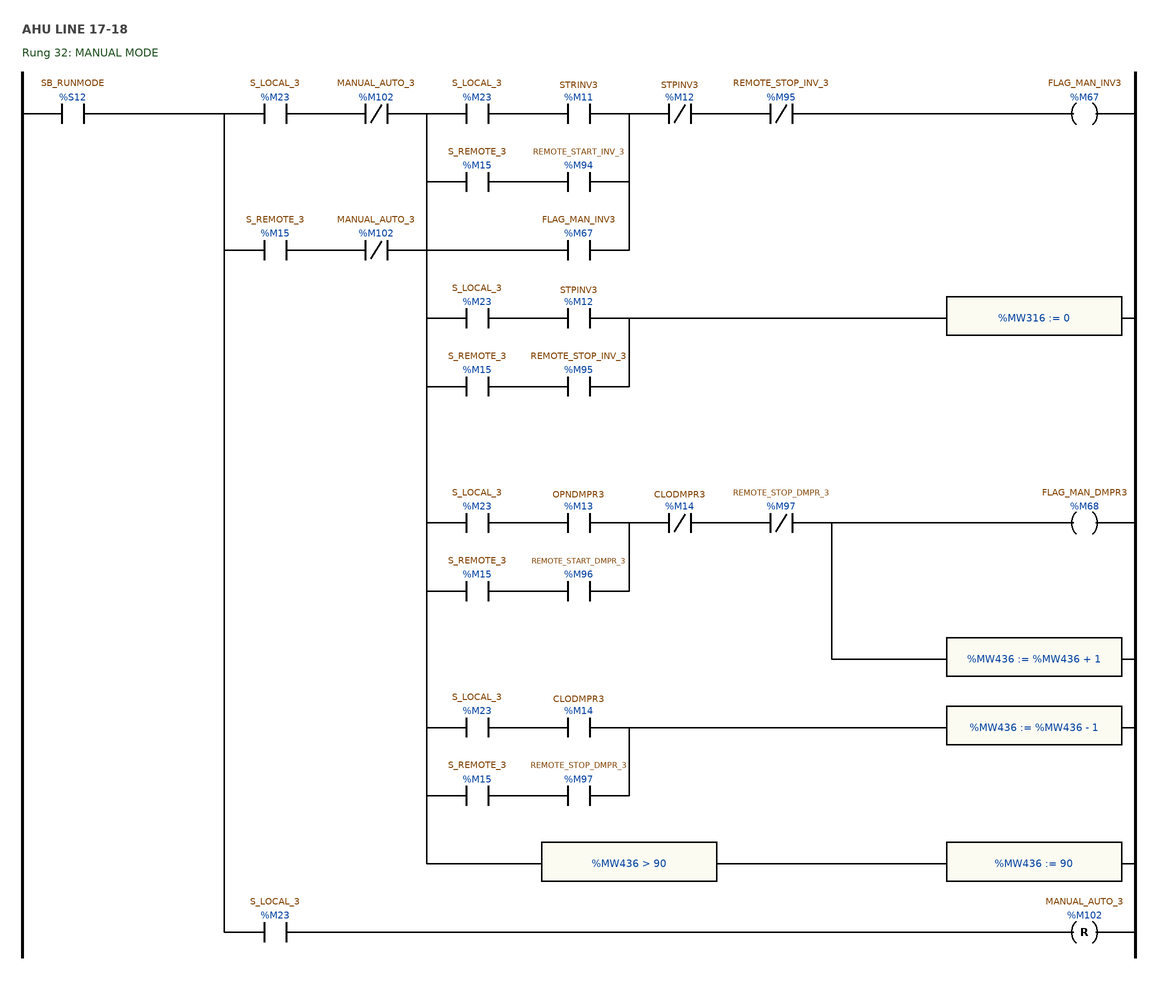

// Rung 32: MANUAL MODE
  LD %S12                 (* SB_RUNMODE *)
  MPS
  AND( %M23               (* S_LOCAL_3 *)
  ANDN %M102              (* MANUAL_AUTO_3 *)
  OR( %M15                (* S_REMOTE_3 *)
  ANDN %M102              (* MANUAL_AUTO_3 *)
  )
  )
  MPS
  AND( %M23               (* S_LOCAL_3 *)
  AND %M11                (* STRINV3 *)
  OR( %M15                (* S_REMOTE_3 *)
  AND %M94                (* REMOTE_START_INV_3 *)
  )
  OR %M67                 (* FLAG_MAN_INV3 *)
  )
  ANDN %M12               (* STPINV3 *)
  ANDN %M95               (* REMOTE_STOP_INV_3 *)
  ST %M67                 (* FLAG_MAN_INV3 *)
  MRD
  AND( %M23               (* S_LOCAL_3 *)
  AND %M12                (* STPINV3 *)
  OR( %M15                (* S_REMOTE_3 *)
  AND %M95                (* REMOTE_STOP_INV_3 *)
  )
  )
  [ %MW316 := 0 ]         (* SET_SPEED_INV_3 *)
  MRD
  AND( %M23               (* S_LOCAL_3 *)
  AND %M13                (* OPNDMPR3 *)
  OR( %M15                (* S_REMOTE_3 *)
  AND %M96                (* REMOTE_START_DMPR_3 *)
  )
  )
  ANDN %M14               (* CLODMPR3 *)
  ANDN %M97               (* REMOTE_STOP_DMPR_3 *)
  ST %M68                 (* FLAG_MAN_DMPR3 *)
  [ %MW436 := %MW436 + 1 ](* SET_DAMPER_3_POSITION, SET_DAMPER_3_POSITION *)
  MRD
  AND( %M23               (* S_LOCAL_3 *)
  AND %M14                (* CLODMPR3 *)
  OR( %M15                (* S_REMOTE_3 *)
  AND %M97                (* REMOTE_STOP_DMPR_3 *)
  )
  )
  [ %MW436 := %MW436 - 1 ](* SET_DAMPER_3_POSITION, SET_DAMPER_3_POSITION *)
  MPP
  AND [ %MW436 > 90 ]     (* SET_DAMPER_3_POSITION *)
  [ %MW436 := 90 ]        (* SET_DAMPER_3_POSITION *)
  MPP
  AND %M23                (* S_LOCAL_3 *)
  R %M102                 (* MANUAL_AUTO_3 *)
  // as ST:
  //   FLAG_MAN_INV3 := SB_RUNMODE AND (S_LOCAL_3 AND NOT MANUAL_AUTO_3 OR S_REMOTE_3 AND NOT MANUAL_AUTO_3) AND (S_LOCAL_3 AND STRINV3 OR S_REMOTE_3 AND REMOTE_START_INV_3 OR FLAG_MAN_INV3) AND NOT STPINV3 AND NOT REMOTE_STOP_INV_3;
  //   IF SB_RUNMODE AND (S_LOCAL_3 AND NOT MANUAL_AUTO_3 OR S_REMOTE_3 AND NOT MANUAL_AUTO_3) AND (S_LOCAL_3 AND STPINV3 OR S_REMOTE_3 AND REMOTE_STOP_INV_3) THEN SET_SPEED_INV_3 := 0; END_IF;
  //   FLAG_MAN_DMPR3 := SB_RUNMODE AND (S_LOCAL_3 AND NOT MANUAL_AUTO_3 OR S_REMOTE_3 AND NOT MANUAL_AUTO_3) AND (S_LOCAL_3 AND OPNDMPR3 OR S_REMOTE_3 AND REMOTE_START_DMPR_3) AND NOT CLODMPR3 AND NOT REMOTE_STOP_DMPR_3;
  //   IF SB_RUNMODE AND (S_LOCAL_3 AND NOT MANUAL_AUTO_3 OR S_REMOTE_3 AND NOT MANUAL_AUTO_3) AND (S_LOCAL_3 AND OPNDMPR3 OR S_REMOTE_3 AND REMOTE_START_DMPR_3) AND NOT CLODMPR3 AND NOT REMOTE_STOP_DMPR_3 THEN SET_DAMPER_3_POSITION := SET_DAMPER_3_POSITION + 1; END_IF;
  //   IF SB_RUNMODE AND (S_LOCAL_3 AND NOT MANUAL_AUTO_3 OR S_REMOTE_3 AND NOT MANUAL_AUTO_3) AND (S_LOCAL_3 AND CLODMPR3 OR S_REMOTE_3 AND REMOTE_STOP_DMPR_3) THEN SET_DAMPER_3_POSITION := SET_DAMPER_3_POSITION - 1; END_IF;
  //   IF SB_RUNMODE AND (S_LOCAL_3 AND NOT MANUAL_AUTO_3 OR S_REMOTE_3 AND NOT MANUAL_AUTO_3) AND SET_DAMPER_3_POSITION > 90 THEN SET_DAMPER_3_POSITION := 90; END_IF;
  //   IF SB_RUNMODE AND S_LOCAL_3 THEN MANUAL_AUTO_3 := FALSE; END_IF;

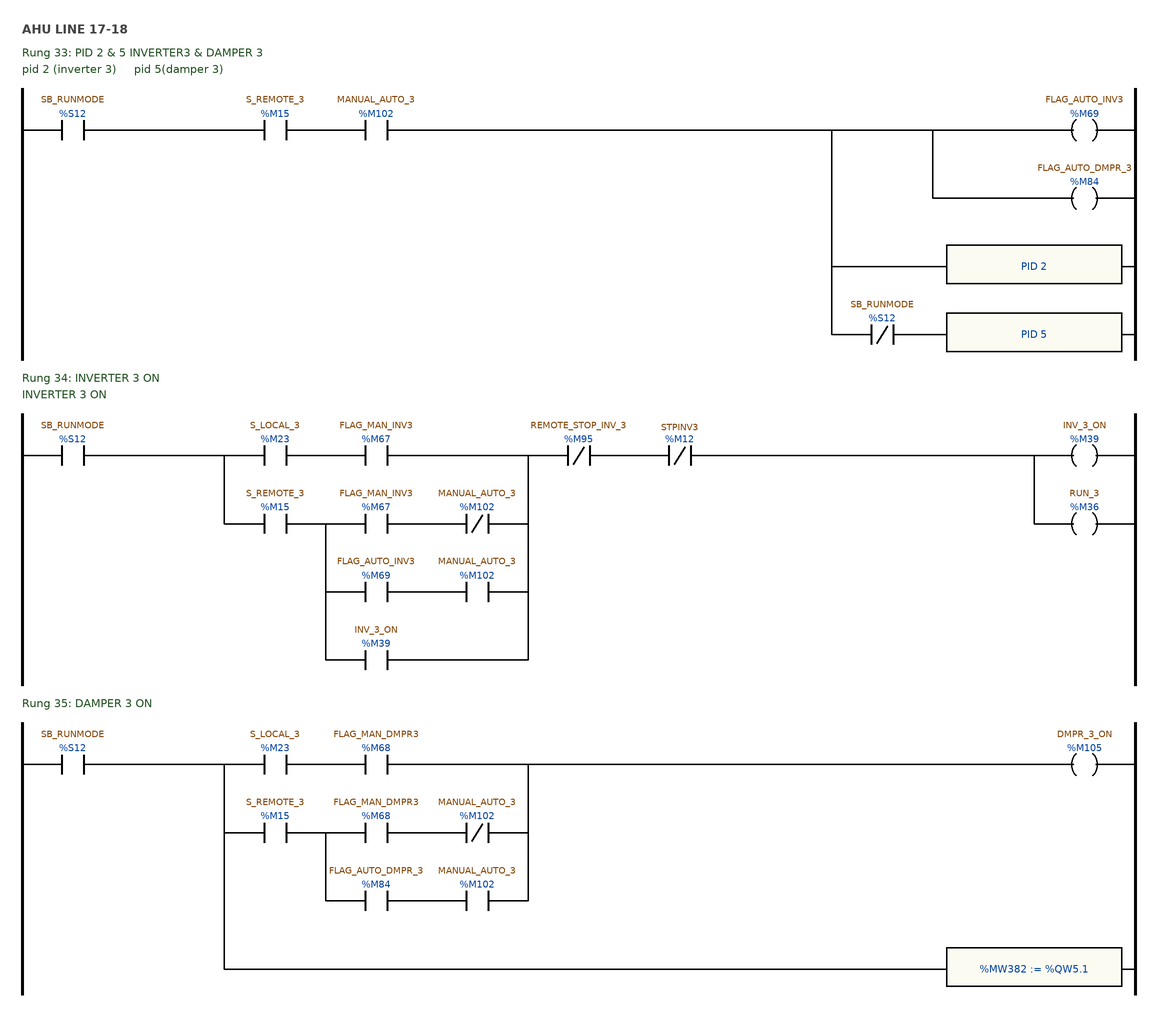

// Rung 33: PID 2 & 5 INVERTER3 & DAMPER 3
// pid 2 (inverter 3)     pid 5(damper 3)
  LD %S12                 (* SB_RUNMODE *)
  AND %M15                (* S_REMOTE_3 *)
  AND %M102               (* MANUAL_AUTO_3 *)
  MPS
  ST %M69                 (* FLAG_AUTO_INV3 *)
  ST %M84                 (* FLAG_AUTO_DMPR_3 *)
  MRD
  [ PID 2 ]
  MPP
  ANDN %S12               (* SB_RUNMODE *)
  [ PID 5 ]
  // as ST:
  //   FLAG_AUTO_INV3 := SB_RUNMODE AND S_REMOTE_3 AND MANUAL_AUTO_3;
  //   FLAG_AUTO_DMPR_3 := SB_RUNMODE AND S_REMOTE_3 AND MANUAL_AUTO_3;
  //   IF SB_RUNMODE AND S_REMOTE_3 AND MANUAL_AUTO_3 THEN PID 2; END_IF;
  //   IF SB_RUNMODE AND S_REMOTE_3 AND MANUAL_AUTO_3 AND NOT SB_RUNMODE THEN PID 5; END_IF;

// Rung 34: INVERTER 3 ON
// INVERTER 3 ON
  LD %S12                 (* SB_RUNMODE *)
  AND( %M23               (* S_LOCAL_3 *)
  AND %M67                (* FLAG_MAN_INV3 *)
  OR( %M15                (* S_REMOTE_3 *)
  AND( %M67               (* FLAG_MAN_INV3 *)
  ANDN %M102              (* MANUAL_AUTO_3 *)
  OR( %M69                (* FLAG_AUTO_INV3 *)
  AND %M102               (* MANUAL_AUTO_3 *)
  )
  OR %M39                 (* INV_3_ON *)
  )
  )
  )
  ANDN %M95               (* REMOTE_STOP_INV_3 *)
  ANDN %M12               (* STPINV3 *)
  ST %M39                 (* INV_3_ON *)
  ST %M36                 (* RUN_3 *)
  // as ST:
  //   _t1 := SB_RUNMODE AND (S_LOCAL_3 AND FLAG_MAN_INV3 OR S_REMOTE_3 AND (FLAG_MAN_INV3 AND NOT MANUAL_AUTO_3 OR FLAG_AUTO_INV3 AND MANUAL_AUTO_3 OR INV_3_ON)) AND NOT REMOTE_STOP_INV_3 AND NOT STPINV3;
  //   INV_3_ON := _t1;
  //   RUN_3 := _t1;

// Rung 35: DAMPER 3 ON
  LD %S12                 (* SB_RUNMODE *)
  MPS
  AND( %M23               (* S_LOCAL_3 *)
  AND %M68                (* FLAG_MAN_DMPR3 *)
  OR( %M15                (* S_REMOTE_3 *)
  AND( %M68               (* FLAG_MAN_DMPR3 *)
  ANDN %M102              (* MANUAL_AUTO_3 *)
  OR( %M84                (* FLAG_AUTO_DMPR_3 *)
  AND %M102               (* MANUAL_AUTO_3 *)
  )
  )
  )
  )
  ST %M105                (* DMPR_3_ON *)
  MPP
  [ %MW382 := %QW5.1 ]    (* DMPR_3_VIEW, AO_DMPR_3 *)
  // as ST:
  //   DMPR_3_ON := SB_RUNMODE AND (S_LOCAL_3 AND FLAG_MAN_DMPR3 OR S_REMOTE_3 AND (FLAG_MAN_DMPR3 AND NOT MANUAL_AUTO_3 OR FLAG_AUTO_DMPR_3 AND MANUAL_AUTO_3));
  //   IF SB_RUNMODE THEN DMPR_3_VIEW := AO_DMPR_3; END_IF;

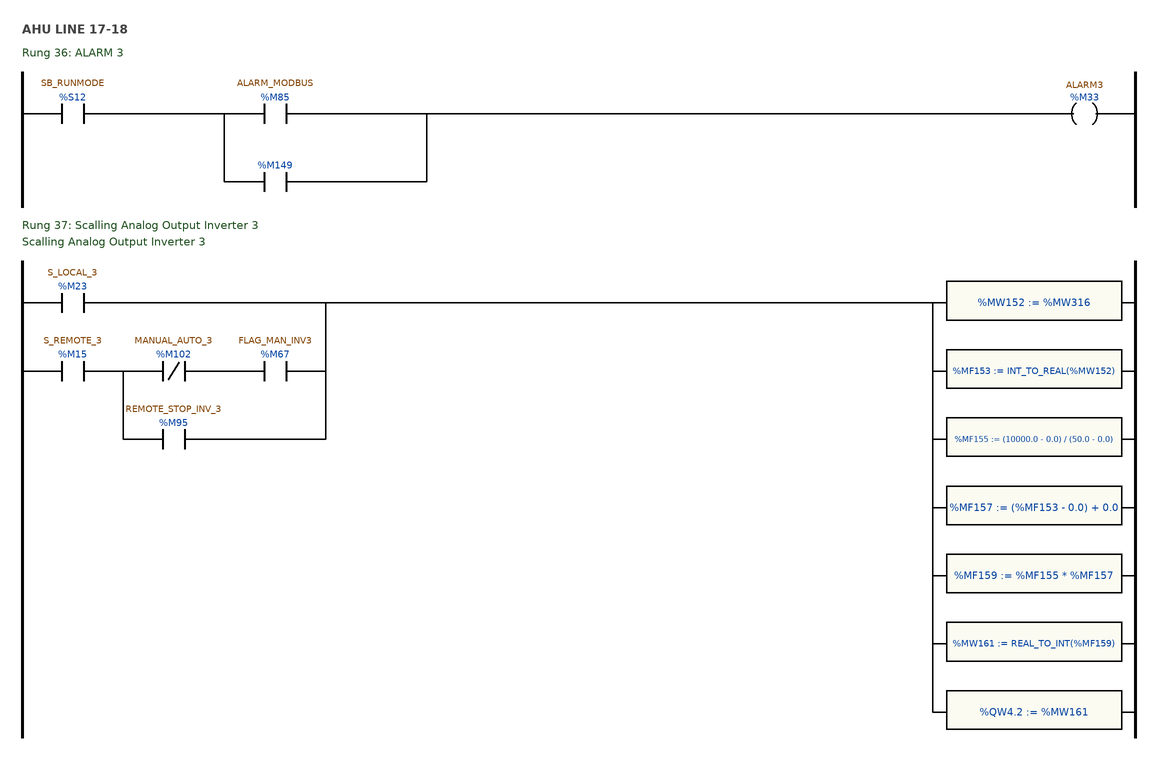

// Rung 36: ALARM 3
  LD %S12                 (* SB_RUNMODE *)
  AND( %M85               (* ALARM_MODBUS *)
  OR %M149
  )
  ST %M33                 (* ALARM3 *)
  // as ST:
  //   ALARM3 := SB_RUNMODE AND (ALARM_MODBUS OR %M149);

// Rung 37: Scalling Analog Output Inverter 3
// Scalling Analog Output Inverter 3
  LD %M23                 (* S_LOCAL_3 *)
  OR( %M15                (* S_REMOTE_3 *)
  AND(N %M102             (* MANUAL_AUTO_3 *)
  AND %M67                (* FLAG_MAN_INV3 *)
  OR %M95                 (* REMOTE_STOP_INV_3 *)
  )
  )
  [ %MW152 := %MW316 ]    (* SET_SPEED_INV_3 *)
  [ %MF153 := INT_TO_REAL ( %MW152 ) ]
  [%MF155 := (10000.0 - 0.0) / (50.0 - 0.0)]
  [%MF157 := (%MF153 - 0.0) + 0.0]
  [ %MF159 := %MF155 * %MF157 ]
  [ %MW161 := REAL_TO_INT ( %MF159 ) ](* AO_SCALE_TEMP_3 *)
  [ %QW4.2 := %MW161 ]    (* AO_INV_3, AO_SCALE_TEMP_3 *)
  // as ST:
  //   IF S_LOCAL_3 OR S_REMOTE_3 AND (NOT MANUAL_AUTO_3 AND FLAG_MAN_INV3 OR REMOTE_STOP_INV_3) THEN %MW152 := SET_SPEED_INV_3; END_IF;
  //   IF S_LOCAL_3 OR S_REMOTE_3 AND (NOT MANUAL_AUTO_3 AND FLAG_MAN_INV3 OR REMOTE_STOP_INV_3) THEN %MF153 := INT_TO_REAL ( %MW152 ); END_IF;
  //   IF S_LOCAL_3 OR S_REMOTE_3 AND (NOT MANUAL_AUTO_3 AND FLAG_MAN_INV3 OR REMOTE_STOP_INV_3) THEN %MF155 := (10000.0 - 0.0) / (50.0 - 0.0); END_IF;
  //   IF S_LOCAL_3 OR S_REMOTE_3 AND (NOT MANUAL_AUTO_3 AND FLAG_MAN_INV3 OR REMOTE_STOP_INV_3) THEN %MF157 := (%MF153 - 0.0) + 0.0; END_IF;
  //   IF S_LOCAL_3 OR S_REMOTE_3 AND (NOT MANUAL_AUTO_3 AND FLAG_MAN_INV3 OR REMOTE_STOP_INV_3) THEN %MF159 := %MF155 * %MF157; END_IF;
  //   IF S_LOCAL_3 OR S_REMOTE_3 AND (NOT MANUAL_AUTO_3 AND FLAG_MAN_INV3 OR REMOTE_STOP_INV_3) THEN AO_SCALE_TEMP_3 := REAL_TO_INT ( %MF159 ); END_IF;
  //   IF S_LOCAL_3 OR S_REMOTE_3 AND (NOT MANUAL_AUTO_3 AND FLAG_MAN_INV3 OR REMOTE_STOP_INV_3) THEN AO_INV_3 := AO_SCALE_TEMP_3; END_IF;

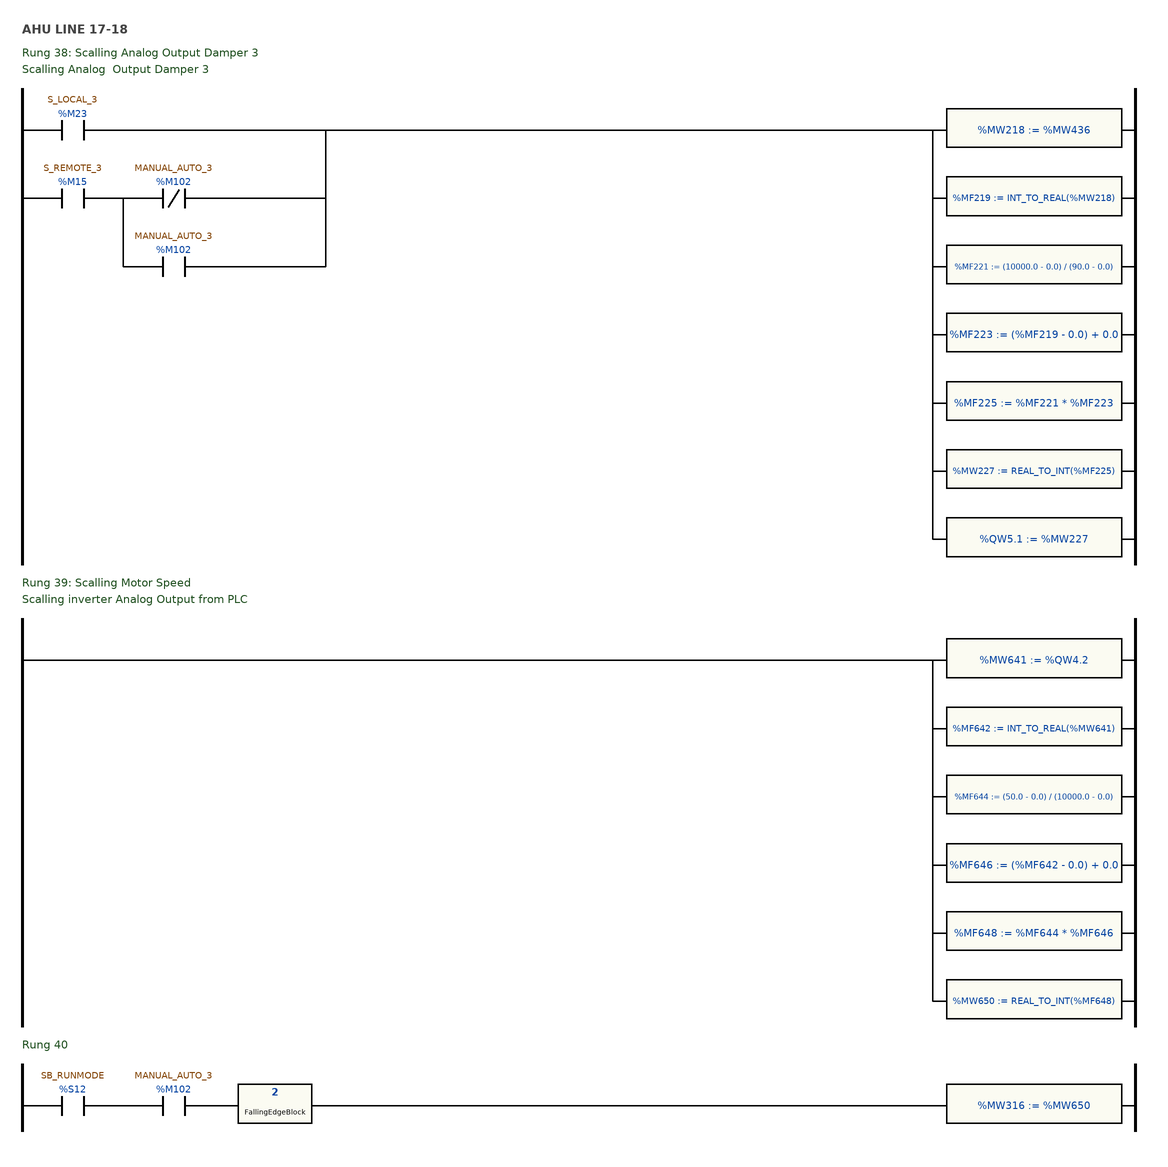

// Rung 38: Scalling Analog Output Damper 3
// Scalling Analog  Output Damper 3
  LD %M23                 (* S_LOCAL_3 *)
  OR( %M15                (* S_REMOTE_3 *)
  AND(N %M102             (* MANUAL_AUTO_3 *)
  OR %M102                (* MANUAL_AUTO_3 *)
  )
  )
  [ %MW218 := %MW436 ]    (* SET_DAMPER_3_POSITION *)
  [ %MF219 := INT_TO_REAL ( %MW218 ) ]
  [%MF221 := (10000.0 - 0.0) / (90.0 - 0.0)]
  [%MF223 := (%MF219 - 0.0) + 0.0]
  [ %MF225 := %MF221 * %MF223 ]
  [ %MW227 := REAL_TO_INT ( %MF225 ) ](* AO_SCALE_HUMIDITY_3 *)
  [ %QW5.1 := %MW227 ]    (* AO_DMPR_3, AO_SCALE_HUMIDITY_3 *)
  // as ST:
  //   IF S_LOCAL_3 OR S_REMOTE_3 AND (NOT MANUAL_AUTO_3 OR MANUAL_AUTO_3) THEN %MW218 := SET_DAMPER_3_POSITION; END_IF;
  //   IF S_LOCAL_3 OR S_REMOTE_3 AND (NOT MANUAL_AUTO_3 OR MANUAL_AUTO_3) THEN %MF219 := INT_TO_REAL ( %MW218 ); END_IF;
  //   IF S_LOCAL_3 OR S_REMOTE_3 AND (NOT MANUAL_AUTO_3 OR MANUAL_AUTO_3) THEN %MF221 := (10000.0 - 0.0) / (90.0 - 0.0); END_IF;
  //   IF S_LOCAL_3 OR S_REMOTE_3 AND (NOT MANUAL_AUTO_3 OR MANUAL_AUTO_3) THEN %MF223 := (%MF219 - 0.0) + 0.0; END_IF;
  //   IF S_LOCAL_3 OR S_REMOTE_3 AND (NOT MANUAL_AUTO_3 OR MANUAL_AUTO_3) THEN %MF225 := %MF221 * %MF223; END_IF;
  //   IF S_LOCAL_3 OR S_REMOTE_3 AND (NOT MANUAL_AUTO_3 OR MANUAL_AUTO_3) THEN AO_SCALE_HUMIDITY_3 := REAL_TO_INT ( %MF225 ); END_IF;
  //   IF S_LOCAL_3 OR S_REMOTE_3 AND (NOT MANUAL_AUTO_3 OR MANUAL_AUTO_3) THEN AO_DMPR_3 := AO_SCALE_HUMIDITY_3; END_IF;

// Rung 39: Scalling Motor Speed
// Scalling inverter Analog Output from PLC
  LD 1
  [ %MW641 := %QW4.2 ]    (* AO_INV_3 *)
  [ %MF642 := INT_TO_REAL ( %MW641 ) ]
  [%MF644 := (50.0 - 0.0) / (10000.0 - 0.0)]
  [%MF646 := (%MF642 - 0.0) + 0.0]
  [ %MF648 := %MF644 * %MF646 ]
  [ %MW650 := REAL_TO_INT ( %MF648 ) ](* INV_3_HZ *)
  // as ST:
  //   %MW641 := AO_INV_3;
  //   %MF642 := INT_TO_REAL ( %MW641 );
  //   %MF644 := (50.0 - 0.0) / (10000.0 - 0.0);
  //   %MF646 := (%MF642 - 0.0) + 0.0;
  //   %MF648 := %MF644 * %MF646;
  //   INV_3_HZ := REAL_TO_INT ( %MF648 );

// Rung 40
  LD %S12                 (* SB_RUNMODE *)
  AND %M102               (* MANUAL_AUTO_3 *)
  FALLING2
  [ %MW316 := %MW650 ]    (* SET_SPEED_INV_3, INV_3_HZ *)
  // as ST:
  //   IF FALLING(SB_RUNMODE AND MANUAL_AUTO_3) THEN SET_SPEED_INV_3 := INV_3_HZ; END_IF;

POU READ WRITE DATA
  (* SectionNumber=5 *)

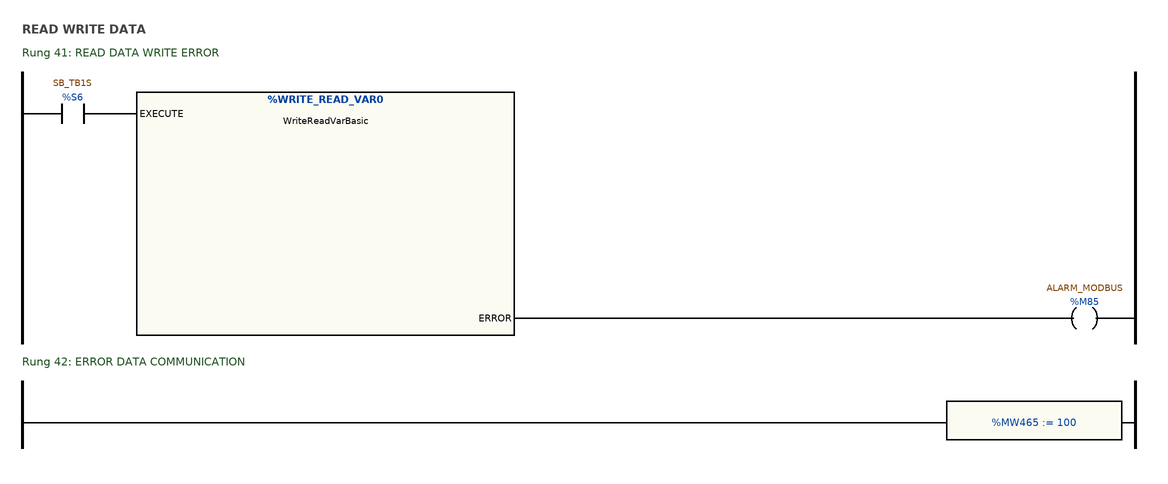

// Rung 41: READ DATA WRITE ERROR
  BLK %WRITE_READ_VAR0
  LD %S6                  (* SB_TB1S *)
  EXECUTE
  OUT_BLK
  LD ERROR
  ST %M85                 (* ALARM_MODBUS *)
  END_BLK
  // as ST:
  //   %WRITE_READ_VAR0(EXECUTE := SB_TB1S);
  //   ALARM_MODBUS := %WRITE_READ_VAR0.ERROR;

// Rung 42: ERROR DATA COMMUNICATION
  LD 1
  [ %MW465 := 100 ]       (* ERROR_DATA *)
  // as ST:
  //   ERROR_DATA := 100;

POU SERIAL DATA
  (* SectionNumber=6 *)

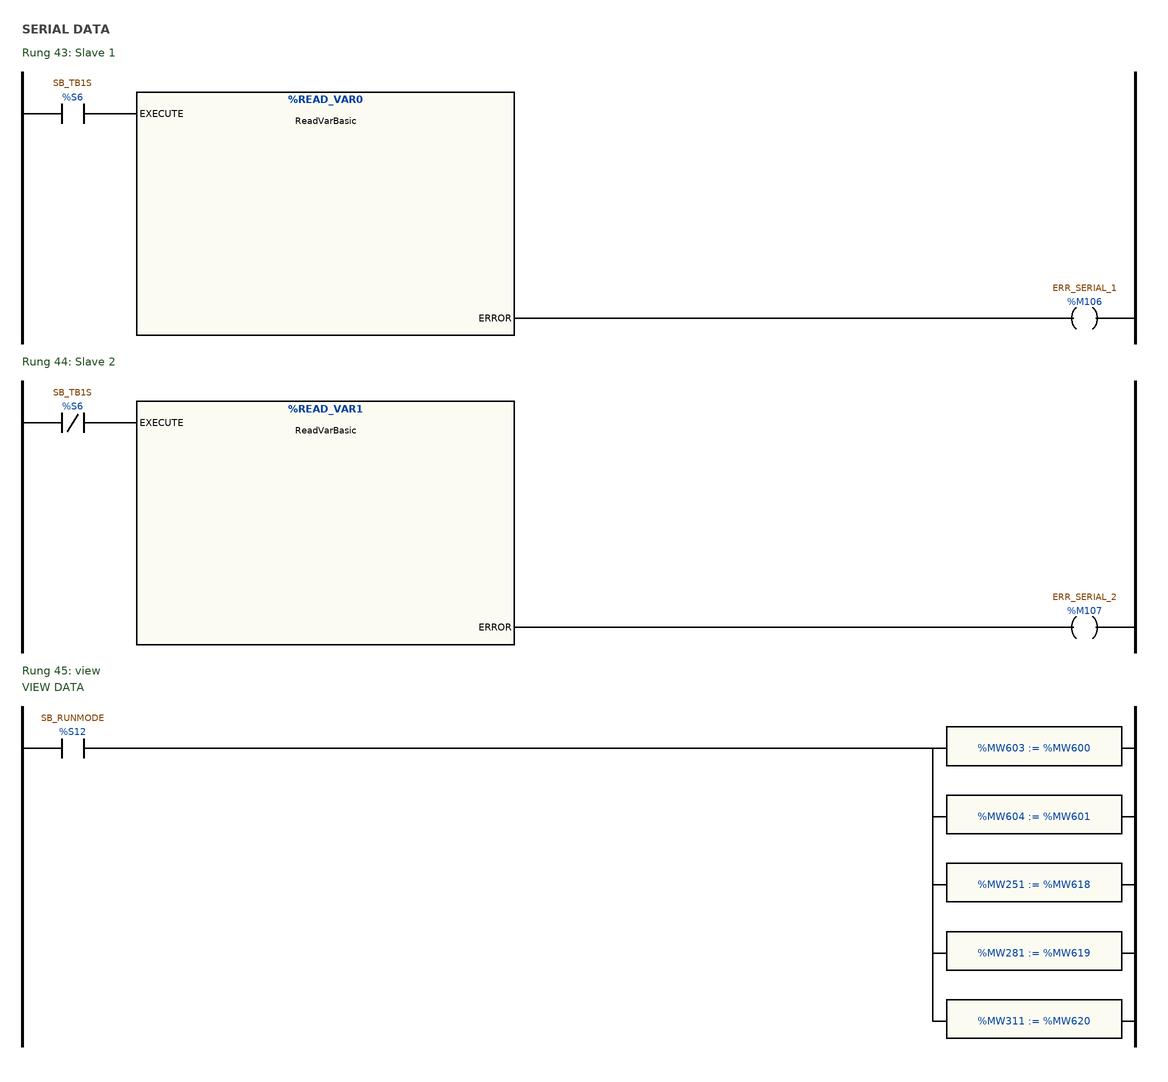

// Rung 43: Slave 1
  BLK %READ_VAR0
  LD %S6                  (* SB_TB1S *)
  EXECUTE
  OUT_BLK
  LD ERROR
  ST %M106                (* ERR_SERIAL_1 *)
  END_BLK
  // as ST:
  //   %READ_VAR0(EXECUTE := SB_TB1S);
  //   ERR_SERIAL_1 := %READ_VAR0.ERROR;

// Rung 44: Slave 2
  BLK %READ_VAR1
  LDN %S6                 (* SB_TB1S *)
  EXECUTE
  OUT_BLK
  LD ERROR
  ST %M107                (* ERR_SERIAL_2 *)
  END_BLK
  // as ST:
  //   %READ_VAR1(EXECUTE := NOT SB_TB1S);
  //   ERR_SERIAL_2 := %READ_VAR1.ERROR;

// Rung 45: view
// VIEW DATA
  LD %S12                 (* SB_RUNMODE *)
  [ %MW603 := %MW600 ]    (* HUMIDITY_LINE_1718 *)
  [ %MW604 := %MW601 ]    (* TEMPERATURE_LINE_1718 *)
  [ %MW251 := %MW618 ]    (* TEMP_1_SETPOINT *)
  [ %MW281 := %MW619 ]    (* TEMP_2_SETPOINT *)
  [ %MW311 := %MW620 ]    (* TEMP_3_SETPOINT *)
  // as ST:
  //   IF SB_RUNMODE THEN %MW603 := HUMIDITY_LINE_1718; END_IF;
  //   IF SB_RUNMODE THEN %MW604 := TEMPERATURE_LINE_1718; END_IF;
  //   IF SB_RUNMODE THEN TEMP_1_SETPOINT := %MW618; END_IF;
  //   IF SB_RUNMODE THEN TEMP_2_SETPOINT := %MW619; END_IF;
  //   IF SB_RUNMODE THEN TEMP_3_SETPOINT := %MW620; END_IF;

POU ALARM CONFIGURATION
  (* SectionNumber=7 *)

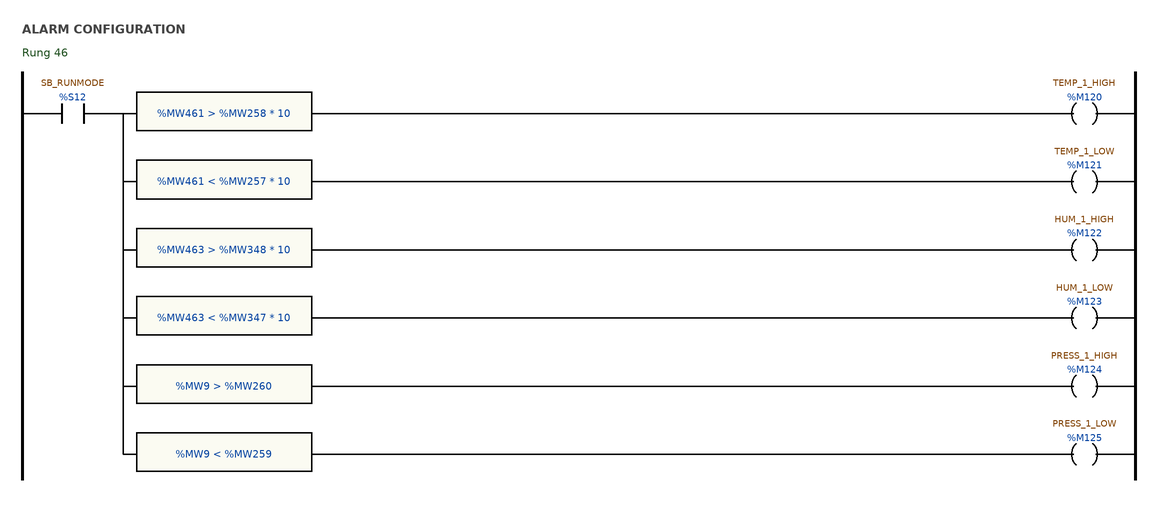

// Rung 46
  LD %S12                 (* SB_RUNMODE *)
  MPS
  AND [%MW461 > %MW258 * 10](* TEMP_1_DATA_SERIAL, ALRM_TEMP1_HIGH_SET *)
  ST %M120                (* TEMP_1_HIGH *)
  MRD
  AND [%MW461 < %MW257 * 10](* TEMP_1_DATA_SERIAL, ALRM_TEMP1_LOW_SET *)
  ST %M121                (* TEMP_1_LOW *)
  MRD
  AND [%MW463 > %MW348 * 10](* HUMIDITY_1_DATA_SERIAL, ALRM_HUMIDITY_1_HIGH_SET *)
  ST %M122                (* HUM_1_HIGH *)
  MRD
  AND [%MW463 < %MW347 * 10](* HUMIDITY_1_DATA_SERIAL, ALRM_HUMIDITY_1_LOW_SET *)
  ST %M123                (* HUM_1_LOW *)
  MRD
  AND [ %MW9 > %MW260 ]   (* AI_SCALE_DIFF_PRESSURE_1, ALRM_PRESS1_HIGH_SET *)
  ST %M124                (* PRESS_1_HIGH *)
  MPP
  AND [ %MW9 < %MW259 ]   (* AI_SCALE_DIFF_PRESSURE_1, ALRM_PRESS1_LOW_SET *)
  ST %M125                (* PRESS_1_LOW *)
  // as ST:
  //   TEMP_1_HIGH := SB_RUNMODE AND TEMP_1_DATA_SERIAL > ALRM_TEMP1_HIGH_SET * 10;
  //   TEMP_1_LOW := SB_RUNMODE AND TEMP_1_DATA_SERIAL < ALRM_TEMP1_LOW_SET * 10;
  //   HUM_1_HIGH := SB_RUNMODE AND HUMIDITY_1_DATA_SERIAL > ALRM_HUMIDITY_1_HIGH_SET * 10;
  //   HUM_1_LOW := SB_RUNMODE AND HUMIDITY_1_DATA_SERIAL < ALRM_HUMIDITY_1_LOW_SET * 10;
  //   PRESS_1_HIGH := SB_RUNMODE AND AI_SCALE_DIFF_PRESSURE_1 > ALRM_PRESS1_HIGH_SET;
  //   PRESS_1_LOW := SB_RUNMODE AND AI_SCALE_DIFF_PRESSURE_1 < ALRM_PRESS1_LOW_SET;

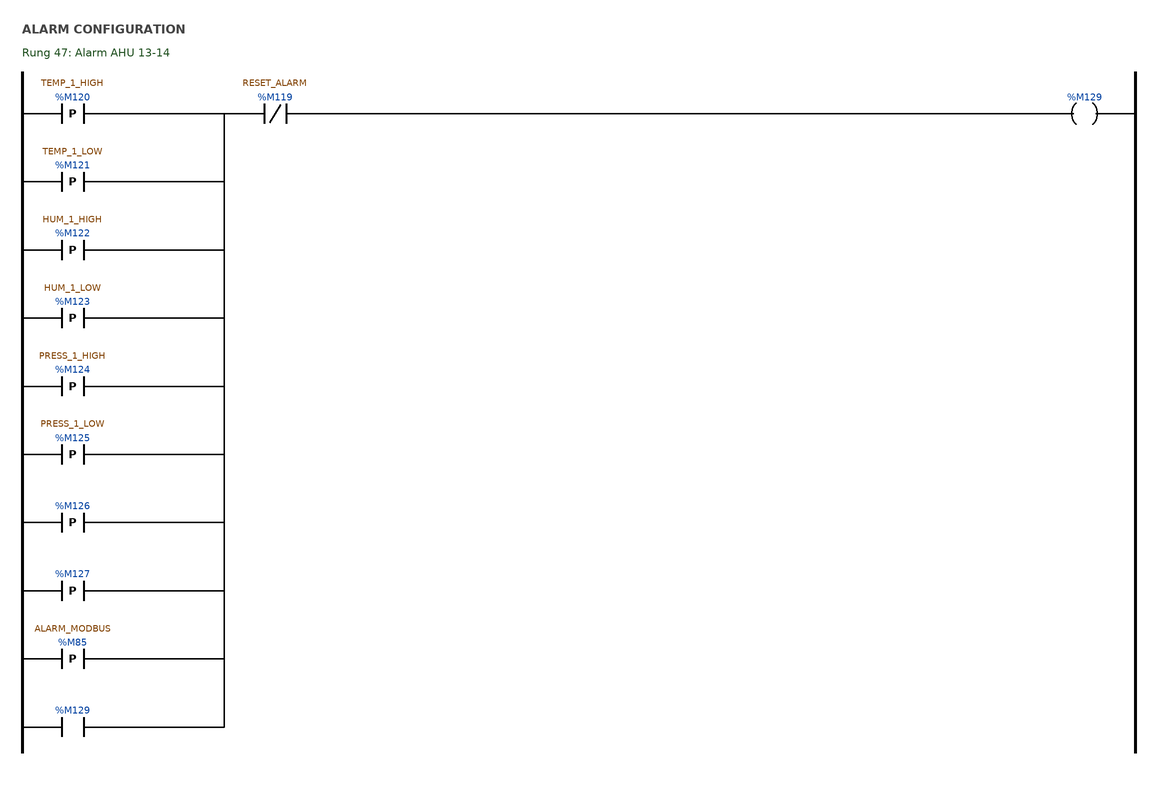

// Rung 47: Alarm AHU 13-14
  LDR %M120               (* TEMP_1_HIGH *)
  ORR %M121               (* TEMP_1_LOW *)
  ORR %M122               (* HUM_1_HIGH *)
  ORR %M123               (* HUM_1_LOW *)
  ORR %M124               (* PRESS_1_HIGH *)
  ORR %M125               (* PRESS_1_LOW *)
  ORR %M126
  ORR %M127
  ORR %M85                (* ALARM_MODBUS *)
  OR %M129
  ANDN %M119              (* RESET_ALARM *)
  ST %M129
  // as ST:
  //   %M129 := (RISING(TEMP_1_HIGH) OR RISING(TEMP_1_LOW) OR RISING(HUM_1_HIGH) OR RISING(HUM_1_LOW) OR RISING(PRESS_1_HIGH) OR RISING(PRESS_1_LOW) OR RISING(%M126) OR RISING(%M127) OR RISING(ALARM_MODBUS) OR %M129) AND NOT RESET_ALARM;

